LIN {X 0,Y 411.222,Z 389.379,A -85,B 0,C 180,E1 -10484.622,E2 -10484.622} C_VEL
LIN {X 0,Y 411.796,Z 392.619,A -85,B 0,C 180,E1 -10487.213,E2 -10487.213} C_VEL
LIN {X 0,Y 412.5,Z 396.68,A -85,B 0,C 180,E1 -10490.059,E2 -10490.059} C_VEL
LIN {X 0,Y 413.335,Z 401.503,A -85,B 0,C 180,E1 -10493.05,E2 -10493.05} C_VEL
LIN {X 0,Y 413.268,Z 404.546,A -85,B 0,C 180,E1 -10494.715,E2 -10494.715} C_VEL
LIN {X 0,Y 412.637,Z 410.141,A -85,B 0,C 180,E1 -10497.559,E2 -10497.559} C_VEL
LIN {X 0,Y 411.855,Z 417.317,A -85,B 0,C 180,E1 -10500.96,E2 -10500.96} C_VEL
LIN {X 0,Y 411.43,Z 424.49,A -85,B 0,C 180,E1 -10504.182,E2 -10504.182} C_VEL
LIN {X 0,Y 410.913,Z 433.22,A -85,B 0,C 180,E1 -10507.902,E2 -10507.902} C_VEL
LIN {X 0,Y 410.581,Z 440.827,A -85,B 0,C 180,E1 -10511.025,E2 -10511.025} C_VEL
LIN {X 0,Y 410.449,Z 443.604,A -85,B 0,C 180,E1 -10512.147,E2 -10512.147} C_VEL
LIN {X 0,Y 412.936,Z 457.87,A -85,B 0,C 180,E1 -10512.764,E2 -10512.764} C_VEL
LIN {X 0,Y 414.283,Z 471.211,A -85,B 0,C 180,E1 -10513.496,E2 -10513.496} C_VEL
LIN {X 0,Y 414.496,Z 479.224,A -85,B 0,C 180,E1 -10514.011,E2 -10514.011} C_VEL
LIN {X 0,Y 413.649,Z 490.528,A -85,B 0,C 180,E1 -10514.861,E2 -10514.861} C_VEL
LIN {X 0,Y 412.726,Z 502.13,A -85,B 0,C 180,E1 -10515.961,E2 -10515.961} C_VEL
LIN {X 0,Y 412.087,Z 510.937,A -85,B 0,C 180,E1 -10516.988,E2 -10516.988} C_VEL
LIN {X 0,Y 411.502,Z 519.45,A -85,B 0,C 180,E1 -10518.178,E2 -10518.178} C_VEL
LIN {X 0,Y 410.835,Z 528.113,A -85,B 0,C 180,E1 -10519.656,E2 -10519.656} C_VEL
LIN {X 0,Y 410.451,Z 535.1,A -85,B 0,C 180,E1 -10521.139,E2 -10521.139} C_VEL
LIN {X 0,Y 410.181,Z 540.719,A -85,B 0,C 180,E1 -10522.621,E2 -10522.621} C_VEL
LIN {X 0,Y 410.036,Z 545.145,A -85,B 0,C 180,E1 -10524.101,E2 -10524.101} C_VEL
LIN {X 0,Y 410.055,Z 547.506,A -85,B 0,C 180,E1 -10525.088,E2 -10525.088} C_VEL
LIN {X 0,Y 409.968,Z 549.385,A -85,B 0,C 180,E1 -10526.072,E2 -10526.072} C_VEL
LIN {X 0,Y 410.023,Z 550.818,A -85,B 0,C 180,E1 -10527.056,E2 -10527.056} C_VEL
LIN {X 0,Y 410.057,Z 551.847,A -85,B 0,C 180,E1 -10528.039,E2 -10528.039} C_VEL
LIN {X 0,Y 410.027,Z 552.471,A -85,B 0,C 180,E1 -10529.022,E2 -10529.022} C_VEL
LIN {X 0,Y 410.034,Z 552.654,A -85,B 0,C 180,E1 -10530.004,E2 -10530.004} C_VEL
LIN {X 0,Y 410.028,Z 552.419,A -85,B 0,C 180,E1 -10530.986,E2 -10530.986} C_VEL
LIN {X 0,Y 410.06,Z 551.791,A -85,B 0,C 180,E1 -10531.968,E2 -10531.968} C_VEL
LIN {X 0,Y 410.055,Z 550.757,A -85,B 0,C 180,E1 -10532.951,E2 -10532.951} C_VEL
LIN {X 0,Y 409.972,Z 549.254,A -85,B 0,C 180,E1 -10533.935,E2 -10533.935} C_VEL
LIN {X 0,Y 410.073,Z 546.197,A -85,B 0,C 180,E1 -10535.412,E2 -10535.412} C_VEL
LIN {X 0,Y 410.168,Z 542.052,A -85,B 0,C 180,E1 -10536.892,E2 -10536.892} C_VEL
LIN {X 0,Y 410.399,Z 535.69,A -85,B 0,C 180,E1 -10538.621,E2 -10538.621} C_VEL
LIN {X 0,Y 410.756,Z 528.758,A -85,B 0,C 180,E1 -10540.104,E2 -10540.104} C_VEL
LIN {X 0,Y 411.348,Z 520.088,A -85,B 0,C 180,E1 -10541.584,E2 -10541.584} C_VEL
LIN {X 0,Y 411.937,Z 511.205,A -85,B 0,C 180,E1 -10542.817,E2 -10542.817} C_VEL
LIN {X 0,Y 412.67,Z 500.31,A -85,B 0,C 180,E1 -10544.048,E2 -10544.048} C_VEL
LIN {X 0,Y 413.369,Z 489.363,A -85,B 0,C 180,E1 -10545.03,E2 -10545.03} C_VEL
LIN {X 0,Y 414.185,Z 477.508,A -85,B 0,C 180,E1 -10545.866,E2 -10545.866} C_VEL
LIN {X 0,Y 414.152,Z 473.913,A -85,B 0,C 180,E1 -10546.087,E2 -10546.087} C_VEL
LIN {X 0,Y 412.627,Z 460.357,A -85,B 0,C 180,E1 -10546.818,E2 -10546.818} C_VEL
LIN {X 0,Y 410.639,Z 447.133,A -85,B 0,C 180,E1 -10547.336,E2 -10547.336} C_VEL
LIN {X 0,Y 410.476,Z 445.601,A -85,B 0,C 180,E1 -10547.387,E2 -10547.387} C_VEL
LIN {X 0,Y 410.779,Z 437.879,A -85,B 0,C 180,E1 -10550.535,E2 -10550.535} C_VEL
LIN {X 0,Y 411.171,Z 430.287,A -85,B 0,C 180,E1 -10553.686,E2 -10553.686} C_VEL
LIN {X 0,Y 411.619,Z 422.72,A -85,B 0,C 180,E1 -10556.887,E2 -10556.887} C_VEL
LIN {X 0,Y 412.336,Z 413.826,A -85,B 0,C 180,E1 -10560.756,E2 -10560.756} C_VEL
LIN {X 0,Y 413.02,Z 406.24,A -85,B 0,C 180,E1 -10564.165,E2 -10564.165} C_VEL
LIN {X 0,Y 413.217,Z 401.187,A -85,B 0,C 180,E1 -10566.536,E2 -10566.536} C_VEL
LIN {X 0,Y 412.171,Z 394.541,A -85,B 0,C 180,E1 -10569.887,E2 -10569.887} C_VEL
LIN {X 0,Y 411.214,Z 389.263,A -85,B 0,C 180,E1 -10572.748,E2 -10572.748} C_VEL
LIN {X 0,Y 411.178,Z 389.268,A -85,B 0,C 180,E1 -10575.883,E2 -10575.883} C_VEL
LIN {X 0,Y 411.163,Z 389.271,A -85,B 0,C 180,E1 -10578.775,E2 -10578.775} C_VEL
LIN {X 0,Y 411.199,Z 389.263,A -85,B 0,C 180,E1 -10582.026,E2 -10582.026} C_VEL
LIN {X 0,Y 411.216,Z 389.265,A -85,B 0,C 180,E1 -10585.124,E2 -10585.124} C_VEL
LIN {X 0,Y 411.178,Z 389.266,A -85,B 0,C 180,E1 -10588.003,E2 -10588.003} C_VEL
LIN {X 0,Y 411.207,Z 389.265,A -85,B 0,C 180,E1 -10591.408,E2 -10591.408} C_VEL
LIN {X 0,Y 411.231,Z 389.263,A -85,B 0,C 180,E1 -10594.933,E2 -10594.933} C_VEL
LIN {X 0,Y 411.218,Z 389.26,A -85,B 0,C 180,E1 -10597.913,E2 -10597.913} C_VEL
LIN {X 0,Y 411.233,Z 389.262,A -85,B 0,C 180,E1 -10601.051,E2 -10601.051} C_VEL
LIN {X 0,Y 411.266,Z 389.255,A -85,B 0,C 180,E1 -10604.131,E2 -10604.131} C_VEL
LIN {X 0,Y 411.316,Z 389.251,A -85,B 0,C 180,E1 -10607.165,E2 -10607.165} C_VEL
LIN {X 0,Y 411.301,Z 389.25,A -85,B 0,C 180,E1 -10610.161,E2 -10610.161} C_VEL
LIN {X 0,Y 411.446,Z 389.236,A -85,B 0,C 180,E1 -10613.132,E2 -10613.132} C_VEL
LIN {X 0,Y 411.314,Z 389.252,A -85,B 0,C 180,E1 -10615.098,E2 -10615.098} C_VEL
LIN {X 0,Y 411.521,Z 389.223,A -85,B 0,C 180,E1 -10618.042,E2 -10618.042} C_VEL
LIN {X 0,Y 411.647,Z 389.208,A -85,B 0,C 180,E1 -10619.999,E2 -10619.999} C_VEL
LIN {X 0,Y 411.457,Z 389.235,A -85,B 0,C 180,E1 -10622.936,E2 -10622.936} C_VEL
LIN {X 0,Y 411.402,Z 389.239,A -85,B 0,C 180,E1 -10626.56,E2 -10626.56} C_VEL
LIN {X 0,Y 411.328,Z 389.25,A -85,B 0,C 180,E1 -10628.845,E2 -10628.845} C_VEL
LIN {X 0,Y 411.291,Z 389.251,A -85,B 0,C 180,E1 -10631.832,E2 -10631.832} C_VEL
LIN {X 0,Y 411.268,Z 389.259,A -85,B 0,C 180,E1 -10634.851,E2 -10634.851} C_VEL
LIN {X 0,Y 411.255,Z 389.257,A -85,B 0,C 180,E1 -10637.914,E2 -10637.914} C_VEL
LIN {X 0,Y 411.205,Z 389.265,A -85,B 0,C 180,E1 -10641.033,E2 -10641.033} C_VEL
LIN {X 0,Y 411.221,Z 389.262,A -85,B 0,C 180,E1 -10644.215,E2 -10644.215} C_VEL
LIN {X 0,Y 411.266,Z 389.254,A -85,B 0,C 180,E1 -10647.476,E2 -10647.476} C_VEL
LIN {X 0,Y 411.197,Z 389.267,A -85,B 0,C 180,E1 -10650.846,E2 -10650.846} C_VEL
LIN {X 0,Y 411.213,Z 389.264,A -85,B 0,C 180,E1 -10654.332,E2 -10654.332} C_VEL
LIN {X 0,Y 411.195,Z 389.265,A -85,B 0,C 180,E1 -10657.972,E2 -10657.972} C_VEL
LIN {X 0,Y 411.164,Z 389.269,A -85,B 0,C 180,E1 -10661.225,E2 -10661.225} C_VEL
LIN {X 0,Y 411.181,Z 389.27,A -85,B 0,C 180,E1 -10664.488,E2 -10664.488} C_VEL
LIN {X 0,Y 411.177,Z 389.268,A -85,B 0,C 180,E1 -10668.191,E2 -10668.191} C_VEL
LIN {X 0,Y 411.212,Z 389.265,A -85,B 0,C 180,E1 -10670.772,E2 -10670.772} C_VEL
LIN {X 0,Y 411.202,Z 389.266,A -85,B 0,C 180,E1 -10674.469,E2 -10674.469} C_VEL
LIN {X 0,Y 411.211,Z 389.263,A -85,B 0,C 180,E1 -10676.871,E2 -10676.871} C_VEL
LIN {X 0,Y 411.235,Z 389.261,A -85,B 0,C 180,E1 -10680.641,E2 -10680.641} C_VEL
LIN {X 0,Y 411.24,Z 389.259,A -85,B 0,C 180,E1 -10683.616,E2 -10683.616} C_VEL
LIN {X 0,Y 411.204,Z 389.265,A -85,B 0,C 180,E1 -10686.849,E2 -10686.849} C_VEL
LIN {X 0,Y 411.215,Z 389.264,A -85,B 0,C 180,E1 -10690.047,E2 -10690.047} C_VEL
LIN {X 0,Y 411.262,Z 389.255,A -85,B 0,C 180,E1 -10693.128,E2 -10693.128} C_VEL
LIN {X 0,Y 411.303,Z 389.25,A -85,B 0,C 180,E1 -10696.893,E2 -10696.893} C_VEL
LIN {X 0,Y 411.29,Z 389.255,A -85,B 0,C 180,E1 -10700.158,E2 -10700.158} C_VEL
LIN {X 0,Y 411.447,Z 389.233,A -85,B 0,C 180,E1 -10703.129,E2 -10703.129} C_VEL
LIN {X 0,Y 411.303,Z 389.25,A -85,B 0,C 180,E1 -10705.095,E2 -10705.095} C_VEL
LIN {X 0,Y 411.506,Z 389.228,A -85,B 0,C 180,E1 -10708.039,E2 -10708.039} C_VEL
LIN {X 0,Y 411.633,Z 389.213,A -85,B 0,C 180,E1 -10709.996,E2 -10709.996} C_VEL
LIN {X 0,Y 411.456,Z 389.231,A -85,B 0,C 180,E1 -10712.934,E2 -10712.934} C_VEL
LIN {X 0,Y 411.45,Z 389.232,A -85,B 0,C 180,E1 -10716.863,E2 -10716.863} C_VEL
LIN {X 0,Y 411.297,Z 389.254,A -85,B 0,C 180,E1 -10719.835,E2 -10719.835} C_VEL
LIN {X 0,Y 411.281,Z 389.253,A -85,B 0,C 180,E1 -10723.301,E2 -10723.301} C_VEL
LIN {X 0,Y 411.247,Z 389.257,A -85,B 0,C 180,E1 -10726.885,E2 -10726.885} C_VEL
LIN {X 0,Y 411.226,Z 389.26,A -85,B 0,C 180,E1 -10727.567,E2 -10727.567} C_VEL
LIN {X 0,Y 410.561,Z 389.346,A -85,B 0,C 180,E1 -10728.385,E2 -10728.385} C_VEL
LIN {X 0,Y 407.673,Z 389.706,A -85,B 0,C 180,E1 -10729.713,E2 -10729.713} C_VEL
LIN {X 0,Y 405.23,Z 390.007,A -85,B 0,C 180,E1 -10730.786,E2 -10730.786} C_VEL
LIN {X 0,Y 404.194,Z 390.138,A -85,B 0,C 180,E1 -10731.616,E2 -10731.616} C_VEL
LIN {X 0,Y 404.118,Z 390.144,A -85,B 0,C 180,E1 -10731.897,E2 -10731.897} C_VEL
LIN {X 0,Y 404.129,Z 390.144,A -85,B 0,C 180,E1 -10735.273,E2 -10735.273} C_VEL
LIN {X 0,Y 403.933,Z 390.172,A -85,B 0,C 180,E1 -10738.014,E2 -10738.014} C_VEL
LIN {X 0,Y 403.533,Z 390.225,A -85,B 0,C 180,E1 -10741.42,E2 -10741.42} C_VEL
LIN {X 0,Y 403.366,Z 390.535,A -85,B 0,C 180,E1 -10742.687,E2 -10742.687} C_VEL
LIN {X 0,Y 403.282,Z 394.125,A -85,B 0,C 180,E1 -10746.33,E2 -10746.33} C_VEL
LIN {X 0,Y 403.206,Z 397.745,A -85,B 0,C 180,E1 -10749.923,E2 -10749.923} C_VEL
LIN {X 0,Y 403.134,Z 400.84,A -85,B 0,C 180,E1 -10752.93,E2 -10752.93} C_VEL
LIN {X 0,Y 403.139,Z 402.439,A -85,B 0,C 180,E1 -10754.466,E2 -10754.466} C_VEL
LIN {X 0,Y 406.744,Z 417.81,A -85,B 0,C 180,E1 -10755.208,E2 -10755.208} C_VEL
LIN {X 0,Y 408.175,Z 425.22,A -85,B 0,C 180,E1 -10755.651,E2 -10755.651} C_VEL
LIN {X 0,Y 407.539,Z 438.082,A -85,B 0,C 180,E1 -10756.481,E2 -10756.481} C_VEL
LIN {X 0,Y 406.786,Z 449.886,A -85,B 0,C 180,E1 -10757.473,E2 -10757.473} C_VEL
LIN {X 0,Y 406.045,Z 460.272,A -85,B 0,C 180,E1 -10758.569,E2 -10758.569} C_VEL
LIN {X 0,Y 405.362,Z 470.406,A -85,B 0,C 180,E1 -10759.891,E2 -10759.891} C_VEL
LIN {X 0,Y 404.616,Z 479.646,A -85,B 0,C 180,E1 -10761.402,E2 -10761.402} C_VEL
LIN {X 0,Y 404.11,Z 486.882,A -85,B 0,C 180,E1 -10762.87,E2 -10762.87} C_VEL
LIN {X 0,Y 403.667,Z 492.658,A -85,B 0,C 180,E1 -10764.322,E2 -10764.322} C_VEL
LIN {X 0,Y 403.332,Z 498.17,A -85,B 0,C 180,E1 -10766.112,E2 -10766.112} C_VEL
LIN {X 0,Y 403.144,Z 502.087,A -85,B 0,C 180,E1 -10767.881,E2 -10767.881} C_VEL
LIN {X 0,Y 402.882,Z 504.621,A -85,B 0,C 180,E1 -10769.611,E2 -10769.611} C_VEL
LIN {X 0,Y 402.866,Z 505.611,A -85,B 0,C 180,E1 -10770.762,E2 -10770.762} C_VEL
LIN {X 0,Y 402.836,Z 506.055,A -85,B 0,C 180,E1 -10771.899,E2 -10771.899} C_VEL
LIN {X 0,Y 402.844,Z 506.017,A -85,B 0,C 180,E1 -10773.027,E2 -10773.027} C_VEL
LIN {X 0,Y 402.925,Z 505.42,A -85,B 0,C 180,E1 -10774.148,E2 -10774.148} C_VEL
LIN {X 0,Y 403.022,Z 504.37,A -85,B 0,C 180,E1 -10775.26,E2 -10775.26} C_VEL
LIN {X 0,Y 403.182,Z 502.794,A -85,B 0,C 180,E1 -10776.365,E2 -10776.365} C_VEL
LIN {X 0,Y 403.485,Z 499.482,A -85,B 0,C 180,E1 -10778.008,E2 -10778.008} C_VEL
LIN {X 0,Y 403.817,Z 494.983,A -85,B 0,C 180,E1 -10779.631,E2 -10779.631} C_VEL
LIN {X 0,Y 404.284,Z 489.17,A -85,B 0,C 180,E1 -10781.241,E2 -10781.241} C_VEL
LIN {X 0,Y 404.982,Z 481.767,A -85,B 0,C 180,E1 -10782.843,E2 -10782.843} C_VEL
LIN {X 0,Y 405.771,Z 472.531,A -85,B 0,C 180,E1 -10784.428,E2 -10784.428} C_VEL
LIN {X 0,Y 406.59,Z 463.669,A -85,B 0,C 180,E1 -10785.655,E2 -10785.655} C_VEL
LIN {X 0,Y 407.379,Z 453.617,A -85,B 0,C 180,E1 -10786.787,E2 -10786.787} C_VEL
LIN {X 0,Y 408.236,Z 442.106,A -85,B 0,C 180,E1 -10787.826,E2 -10787.826} C_VEL
LIN {X 0,Y 409.002,Z 430.403,A -85,B 0,C 180,E1 -10788.654,E2 -10788.654} C_VEL
LIN {X 0,Y 408.992,Z 425.264,A -85,B 0,C 180,E1 -10788.967,E2 -10788.967} C_VEL
LIN {X 0,Y 406.264,Z 413.927,A -85,B 0,C 180,E1 -10789.676,E2 -10789.676} C_VEL
LIN {X 0,Y 403.487,Z 404.713,A -85,B 0,C 180,E1 -10790.192,E2 -10790.192} C_VEL
LIN {X 0,Y 403.71,Z 401.288,A -85,B 0,C 180,E1 -10794.005,E2 -10794.005} C_VEL
LIN {X 0,Y 403.728,Z 399.563,A -85,B 0,C 180,E1 -10796.008,E2 -10796.008} C_VEL
LIN {X 0,Y 404.089,Z 396.193,A -85,B 0,C 180,E1 -10800.001,E2 -10800.001} C_VEL
LIN {X 0,Y 404.245,Z 395.339,A -85,B 0,C 180,E1 -10800.997,E2 -10800.997} C_VEL
LIN {X 0,Y 404.385,Z 391.459,A -85,B 0,C 180,E1 -10805.986,E2 -10805.986} C_VEL
LIN {X 0,Y 404.308,Z 390.129,A -85,B 0,C 180,E1 -10807.994,E2 -10807.994} C_VEL
LIN {X 0,Y 404.244,Z 390.132,A -85,B 0,C 180,E1 -10811.026,E2 -10811.026} C_VEL
LIN {X 0,Y 404.185,Z 390.139,A -85,B 0,C 180,E1 -10814.09,E2 -10814.09} C_VEL
LIN {X 0,Y 404.215,Z 390.135,A -85,B 0,C 180,E1 -10817.193,E2 -10817.193} C_VEL
LIN {X 0,Y 404.175,Z 390.141,A -85,B 0,C 180,E1 -10820.352,E2 -10820.352} C_VEL
LIN {X 0,Y 404.153,Z 390.144,A -85,B 0,C 180,E1 -10823.576,E2 -10823.576} C_VEL
LIN {X 0,Y 404.166,Z 390.143,A -85,B 0,C 180,E1 -10826.88,E2 -10826.88} C_VEL
LIN {X 0,Y 404.124,Z 390.146,A -85,B 0,C 180,E1 -10830.288,E2 -10830.288} C_VEL
LIN {X 0,Y 404.118,Z 390.147,A -85,B 0,C 180,E1 -10833.816,E2 -10833.816} C_VEL
LIN {X 0,Y 404.115,Z 390.148,A -85,B 0,C 180,E1 -10836.88,E2 -10836.88} C_VEL
LIN {X 0,Y 404.145,Z 390.145,A -85,B 0,C 180,E1 -10840.087,E2 -10840.087} C_VEL
LIN {X 0,Y 404.177,Z 390.142,A -85,B 0,C 180,E1 -10843.095,E2 -10843.095} C_VEL
LIN {X 0,Y 404.196,Z 390.36,A -85,B 0,C 180,E1 -10844.068,E2 -10844.068} C_VEL
LIN {X 0,Y 404.794,Z 393.632,A -85,B 0,C 180,E1 -10846.82,E2 -10846.82} C_VEL
LIN {X 0,Y 405.583,Z 398.22,A -85,B 0,C 180,E1 -10850.129,E2 -10850.129} C_VEL
LIN {X 0,Y 406.281,Z 402.362,A -85,B 0,C 180,E1 -10852.745,E2 -10852.745} C_VEL
LIN {X 0,Y 406.355,Z 405.193,A -85,B 0,C 180,E1 -10854.379,E2 -10854.379} C_VEL
LIN {X 0,Y 405.622,Z 411.222,A -85,B 0,C 180,E1 -10857.518,E2 -10857.518} C_VEL
LIN {X 0,Y 404.824,Z 418.276,A -85,B 0,C 180,E1 -10860.921,E2 -10860.921} C_VEL
LIN {X 0,Y 404.355,Z 425.515,A -85,B 0,C 180,E1 -10864.25,E2 -10864.25} C_VEL
LIN {X 0,Y 403.836,Z 434.203,A -85,B 0,C 180,E1 -10868.032,E2 -10868.032} C_VEL
LIN {X 0,Y 403.483,Z 441.762,A -85,B 0,C 180,E1 -10871.206,E2 -10871.206} C_VEL
LIN {X 0,Y 403.41,Z 443.174,A -85,B 0,C 180,E1 -10871.785,E2 -10871.785} C_VEL
LIN {X 0,Y 405.975,Z 457.317,A -85,B 0,C 180,E1 -10872.405,E2 -10872.405} C_VEL
LIN {X 0,Y 407.331,Z 470.431,A -85,B 0,C 180,E1 -10873.142,E2 -10873.142} C_VEL
LIN {X 0,Y 407.68,Z 479.312,A -85,B 0,C 180,E1 -10873.736,E2 -10873.736} C_VEL
LIN {X 0,Y 406.677,Z 491.865,A -85,B 0,C 180,E1 -10874.724,E2 -10874.724} C_VEL
LIN {X 0,Y 405.729,Z 503.121,A -85,B 0,C 180,E1 -10875.842,E2 -10875.842} C_VEL
LIN {X 0,Y 405.047,Z 512.296,A -85,B 0,C 180,E1 -10876.968,E2 -10876.968} C_VEL
LIN {X 0,Y 404.412,Z 520.76,A -85,B 0,C 180,E1 -10878.222,E2 -10878.222} C_VEL
LIN {X 0,Y 403.739,Z 529.089,A -85,B 0,C 180,E1 -10879.726,E2 -10879.726} C_VEL
LIN {X 0,Y 403.34,Z 535.833,A -85,B 0,C 180,E1 -10881.234,E2 -10881.234} C_VEL
LIN {X 0,Y 403.074,Z 541.994,A -85,B 0,C 180,E1 -10882.993,E2 -10882.993} C_VEL
LIN {X 0,Y 402.939,Z 546.023,A -85,B 0,C 180,E1 -10884.499,E2 -10884.499} C_VEL
LIN {X 0,Y 402.887,Z 549.004,A -85,B 0,C 180,E1 -10886.003,E2 -10886.003} C_VEL
LIN {X 0,Y 402.922,Z 550.43,A -85,B 0,C 180,E1 -10887.004,E2 -10887.004} C_VEL
LIN {X 0,Y 402.984,Z 551.453,A -85,B 0,C 180,E1 -10888.005,E2 -10888.005} C_VEL
LIN {X 0,Y 402.95,Z 552.07,A -85,B 0,C 180,E1 -10889.004,E2 -10889.004} C_VEL
LIN {X 0,Y 402.953,Z 552.239,A -85,B 0,C 180,E1 -10890.004,E2 -10890.004} C_VEL
LIN {X 0,Y 402.95,Z 551.998,A -85,B 0,C 180,E1 -10891.003,E2 -10891.003} C_VEL
LIN {X 0,Y 402.988,Z 551.362,A -85,B 0,C 180,E1 -10892.002,E2 -10892.002} C_VEL
LIN {X 0,Y 402.955,Z 550.314,A -85,B 0,C 180,E1 -10893.003,E2 -10893.003} C_VEL
LIN {X 0,Y 402.892,Z 548.795,A -85,B 0,C 180,E1 -10894.005,E2 -10894.005} C_VEL
LIN {X 0,Y 402.97,Z 545.715,A -85,B 0,C 180,E1 -10895.508,E2 -10895.508} C_VEL
LIN {X 0,Y 403.08,Z 541.545,A -85,B 0,C 180,E1 -10897.014,E2 -10897.014} C_VEL
LIN {X 0,Y 403.35,Z 535.158,A -85,B 0,C 180,E1 -10898.773,E2 -10898.773} C_VEL
LIN {X 0,Y 403.708,Z 528.192,A -85,B 0,C 180,E1 -10900.282,E2 -10900.282} C_VEL
LIN {X 0,Y 404.361,Z 519.472,A -85,B 0,C 180,E1 -10901.787,E2 -10901.787} C_VEL
LIN {X 0,Y 405.094,Z 509.107,A -85,B 0,C 180,E1 -10903.226,E2 -10903.226} C_VEL
LIN {X 0,Y 405.807,Z 498.299,A -85,B 0,C 180,E1 -10904.419,E2 -10904.419} C_VEL
LIN {X 0,Y 406.626,Z 487.004,A -85,B 0,C 180,E1 -10905.414,E2 -10905.414} C_VEL
LIN {X 0,Y 407.316,Z 476.778,A -85,B 0,C 180,E1 -10906.13,E2 -10906.13} C_VEL
LIN {X 0,Y 406.271,Z 465.644,A -85,B 0,C 180,E1 -10906.798,E2 -10906.798} C_VEL
LIN {X 0,Y 404.578,Z 452.694,A -85,B 0,C 180,E1 -10907.394,E2 -10907.394} C_VEL
LIN {X 0,Y 403.411,Z 445.239,A -85,B 0,C 180,E1 -10907.672,E2 -10907.672} C_VEL
LIN {X 0,Y 403.747,Z 437.475,A -85,B 0,C 180,E1 -10910.91,E2 -10910.91} C_VEL
LIN {X 0,Y 404.157,Z 429.886,A -85,B 0,C 180,E1 -10914.123,E2 -10914.123} C_VEL
LIN {X 0,Y 404.686,Z 421.74,A -85,B 0,C 180,E1 -10917.662,E2 -10917.662} C_VEL
LIN {X 0,Y 405.388,Z 413.487,A -85,B 0,C 180,E1 -10921.342,E2 -10921.342} C_VEL
LIN {X 0,Y 406.149,Z 405.933,A -85,B 0,C 180,E1 -10924.825,E2 -10924.825} C_VEL
LIN {X 0,Y 406.202,Z 402.199,A -85,B 0,C 180,E1 -10926.622,E2 -10926.622} C_VEL
LIN {X 0,Y 405.181,Z 395.773,A -85,B 0,C 180,E1 -10929.928,E2 -10929.928} C_VEL
LIN {X 0,Y 404.181,Z 390.139,A -85,B 0,C 180,E1 -10933.087,E2 -10933.087} C_VEL
LIN {X 0,Y 404.159,Z 390.143,A -85,B 0,C 180,E1 -10935.927,E2 -10935.927} C_VEL
LIN {X 0,Y 404.118,Z 390.148,A -85,B 0,C 180,E1 -10938.634,E2 -10938.634} C_VEL
LIN {X 0,Y 404.154,Z 390.143,A -85,B 0,C 180,E1 -10941.496,E2 -10941.496} C_VEL
LIN {X 0,Y 404.188,Z 390.139,A -85,B 0,C 180,E1 -10944.983,E2 -10944.983} C_VEL
LIN {X 0,Y 404.152,Z 390.142,A -85,B 0,C 180,E1 -10948.443,E2 -10948.443} C_VEL
LIN {X 0,Y 404.17,Z 390.142,A -85,B 0,C 180,E1 -10950.863,E2 -10950.863} C_VEL
LIN {X 0,Y 404.158,Z 390.139,A -85,B 0,C 180,E1 -10954.231,E2 -10954.231} C_VEL
LIN {X 0,Y 404.182,Z 390.138,A -85,B 0,C 180,E1 -10957.508,E2 -10957.508} C_VEL
LIN {X 0,Y 404.176,Z 390.141,A -85,B 0,C 180,E1 -10960.707,E2 -10960.707} C_VEL
LIN {X 0,Y 404.234,Z 390.131,A -85,B 0,C 180,E1 -10963.848,E2 -10963.848} C_VEL
LIN {X 0,Y 404.297,Z 390.127,A -85,B 0,C 180,E1 -10966.939,E2 -10966.939} C_VEL
LIN {X 0,Y 404.267,Z 390.126,A -85,B 0,C 180,E1 -10969.988,E2 -10969.988} C_VEL
LIN {X 0,Y 404.396,Z 390.114,A -85,B 0,C 180,E1 -10973.012,E2 -10973.012} C_VEL
LIN {X 0,Y 404.285,Z 390.128,A -85,B 0,C 180,E1 -10975.013,E2 -10975.013} C_VEL
LIN {X 0,Y 404.49,Z 390.098,A -85,B 0,C 180,E1 -10978.008,E2 -10978.008} C_VEL
LIN {X 0,Y 404.616,Z 390.083,A -85,B 0,C 180,E1 -10979.999,E2 -10979.999} C_VEL
LIN {X 0,Y 404.416,Z 390.111,A -85,B 0,C 180,E1 -10982.988,E2 -10982.988} C_VEL
LIN {X 0,Y 404.354,Z 390.116,A -85,B 0,C 180,E1 -10986.556,E2 -10986.556} C_VEL
LIN {X 0,Y 404.275,Z 390.129,A -85,B 0,C 180,E1 -10989,E2 -10989} C_VEL
LIN {X 0,Y 404.265,Z 390.127,A -85,B 0,C 180,E1 -10992.04,E2 -10992.04} C_VEL
LIN {X 0,Y 404.214,Z 390.135,A -85,B 0,C 180,E1 -10995.117,E2 -10995.117} C_VEL
LIN {X 0,Y 404.214,Z 390.135,A -85,B 0,C 180,E1 -10998.237,E2 -10998.237} C_VEL
LIN {X 0,Y 404.147,Z 390.142,A -85,B 0,C 180,E1 -11001.418,E2 -11001.418} C_VEL
LIN {X 0,Y 404.179,Z 390.141,A -85,B 0,C 180,E1 -11004.664,E2 -11004.664} C_VEL
LIN {X 0,Y 404.202,Z 390.134,A -85,B 0,C 180,E1 -11007.998,E2 -11007.998} C_VEL
LIN {X 0,Y 404.147,Z 390.141,A -85,B 0,C 180,E1 -11011.556,E2 -11011.556} C_VEL
LIN {X 0,Y 404.191,Z 390.138,A -85,B 0,C 180,E1 -11015.014,E2 -11015.014} C_VEL
LIN {X 0,Y 404.153,Z 390.145,A -85,B 0,C 180,E1 -11018.756,E2 -11018.756} C_VEL
LIN {X 0,Y 404.123,Z 390.145,A -85,B 0,C 180,E1 -11021.596,E2 -11021.596} C_VEL
LIN {X 0,Y 404.15,Z 390.145,A -85,B 0,C 180,E1 -11024.519,E2 -11024.519} C_VEL
LIN {X 0,Y 404.137,Z 390.143,A -85,B 0,C 180,E1 -11027.292,E2 -11027.292} C_VEL
LIN {X 0,Y 404.159,Z 390.142,A -85,B 0,C 180,E1 -11029.951,E2 -11029.951} C_VEL
LIN {X 0,Y 404.14,Z 390.143,A -85,B 0,C 180,E1 -11033.123,E2 -11033.123} C_VEL
LIN {X 0,Y 404.149,Z 390.144,A -85,B 0,C 180,E1 -11036.185,E2 -11036.185} C_VEL
LIN {X 0,Y 404.148,Z 390.142,A -85,B 0,C 180,E1 -11039.712,E2 -11039.712} C_VEL
LIN {X 0,Y 404.197,Z 390.136,A -85,B 0,C 180,E1 -11043.12,E2 -11043.12} C_VEL
LIN {X 0,Y 404.178,Z 390.137,A -85,B 0,C 180,E1 -11045.331,E2 -11045.331} C_VEL
LIN {X 0,Y 404.139,Z 390.145,A -85,B 0,C 180,E1 -11048.577,E2 -11048.577} C_VEL
LIN {X 0,Y 404.209,Z 390.135,A -85,B 0,C 180,E1 -11051.759,E2 -11051.759} C_VEL
LIN {X 0,Y 404.204,Z 390.136,A -85,B 0,C 180,E1 -11054.879,E2 -11054.879} C_VEL
LIN {X 0,Y 404.254,Z 390.131,A -85,B 0,C 180,E1 -11057.955,E2 -11057.955} C_VEL
LIN {X 0,Y 404.4,Z 390.114,A -85,B 0,C 180,E1 -11062.126,E2 -11062.126} C_VEL
LIN {X 0,Y 404.414,Z 390.111,A -85,B 0,C 180,E1 -11064.011,E2 -11064.011} C_VEL
LIN {X 0,Y 404.474,Z 390.104,A -85,B 0,C 180,E1 -11068.005,E2 -11068.005} C_VEL
LIN {X 0,Y 404.602,Z 390.088,A -85,B 0,C 180,E1 -11069.996,E2 -11069.996} C_VEL
LIN {X 0,Y 404.413,Z 390.108,A -85,B 0,C 180,E1 -11072.985,E2 -11072.985} C_VEL
LIN {X 0,Y 404.401,Z 390.11,A -85,B 0,C 180,E1 -11076.984,E2 -11076.984} C_VEL
LIN {X 0,Y 404.26,Z 390.131,A -85,B 0,C 180,E1 -11080.008,E2 -11080.008} C_VEL
LIN {X 0,Y 404.252,Z 390.128,A -85,B 0,C 180,E1 -11083.208,E2 -11083.208} C_VEL
LIN {X 0,Y 404.203,Z 390.134,A -85,B 0,C 180,E1 -11087.005,E2 -11087.005} C_VEL
LIN {X 0,Y 404.146,Z 390.143,A -85,B 0,C 180,E1 -11090.348,E2 -11090.348} C_VEL
LIN {X 0,Y 404.118,Z 390.144,A -85,B 0,C 180,E1 -11091.897,E2 -11091.897} C_VEL
LIN {X 0,Y 403.479,Z 390.227,A -85,B 0,C 180,E1 -11092.729,E2 -11092.729} C_VEL
LIN {X 0,Y 400.657,Z 390.584,A -85,B 0,C 180,E1 -11094.08,E2 -11094.08} C_VEL
LIN {X 0,Y 398.229,Z 390.887,A -85,B 0,C 180,E1 -11095.172,E2 -11095.172} C_VEL
LIN {X 0,Y 397.149,Z 391.018,A -85,B 0,C 180,E1 -11096.015,E2 -11096.015} C_VEL
LIN {X 0,Y 397.041,Z 391.029,A -85,B 0,C 180,E1 -11096.301,E2 -11096.301} C_VEL
LIN {X 0,Y 396.843,Z 391.053,A -85,B 0,C 180,E1 -11098.56,E2 -11098.56} C_VEL
LIN {X 0,Y 396.43,Z 391.11,A -85,B 0,C 180,E1 -11101.687,E2 -11101.687} C_VEL
LIN {X 0,Y 396.368,Z 391.116,A -85,B 0,C 180,E1 -11102.13,E2 -11102.13} C_VEL
LIN {X 0,Y 396.3,Z 392.105,A -85,B 0,C 180,E1 -11103.542,E2 -11103.542} C_VEL
LIN {X 0,Y 396.185,Z 395.575,A -85,B 0,C 180,E1 -11107.089,E2 -11107.089} C_VEL
LIN {X 0,Y 396.134,Z 398.772,A -85,B 0,C 180,E1 -11110.283,E2 -11110.283} C_VEL
LIN {X 0,Y 396.04,Z 402.377,A -85,B 0,C 180,E1 -11113.788,E2 -11113.788} C_VEL
LIN {X 0,Y 396.086,Z 402.806,A -85,B 0,C 180,E1 -11114.198,E2 -11114.198} C_VEL
LIN {X 0,Y 399.463,Z 417.152,A -85,B 0,C 180,E1 -11114.892,E2 -11114.892} C_VEL
LIN {X 0,Y 401.26,Z 425.862,A -85,B 0,C 180,E1 -11115.423,E2 -11115.423} C_VEL
LIN {X 0,Y 400.628,Z 438.667,A -85,B 0,C 180,E1 -11116.268,E2 -11116.268} C_VEL
LIN {X 0,Y 399.882,Z 450.105,A -85,B 0,C 180,E1 -11117.247,E2 -11117.247} C_VEL
LIN {X 0,Y 399.007,Z 461.638,A -85,B 0,C 180,E1 -11118.494,E2 -11118.494} C_VEL
LIN {X 0,Y 398.449,Z 469.984,A -85,B 0,C 180,E1 -11119.607,E2 -11119.607} C_VEL
LIN {X 0,Y 397.709,Z 478.791,A -85,B 0,C 180,E1 -11121.027,E2 -11121.027} C_VEL
LIN {X 0,Y 397.131,Z 486.57,A -85,B 0,C 180,E1 -11122.594,E2 -11122.594} C_VEL
LIN {X 0,Y 396.621,Z 493.007,A -85,B 0,C 180,E1 -11124.216,E2 -11124.216} C_VEL
LIN {X 0,Y 396.293,Z 498.425,A -85,B 0,C 180,E1 -11125.992,E2 -11125.992} C_VEL
LIN {X 0,Y 396.067,Z 502.472,A -85,B 0,C 180,E1 -11127.838,E2 -11127.838} C_VEL
LIN {X 0,Y 395.867,Z 504.336,A -85,B 0,C 180,E1 -11129.014,E2 -11129.014} C_VEL
LIN {X 0,Y 395.797,Z 505.804,A -85,B 0,C 180,E1 -11130.456,E2 -11130.456} C_VEL
LIN {X 0,Y 395.748,Z 506.325,A -85,B 0,C 180,E1 -11131.349,E2 -11131.349} C_VEL
LIN {X 0,Y 395.768,Z 506.495,A -85,B 0,C 180,E1 -11132.598,E2 -11132.598} C_VEL
LIN {X 0,Y 395.788,Z 506.199,A -85,B 0,C 180,E1 -11133.647,E2 -11133.647} C_VEL
LIN {X 0,Y 395.901,Z 505.316,A -85,B 0,C 180,E1 -11134.857,E2 -11134.857} C_VEL
LIN {X 0,Y 396.021,Z 504.067,A -85,B 0,C 180,E1 -11135.911,E2 -11135.911} C_VEL
LIN {X 0,Y 396.26,Z 501.855,A -85,B 0,C 180,E1 -11137.245,E2 -11137.245} C_VEL
LIN {X 0,Y 396.56,Z 498.579,A -85,B 0,C 180,E1 -11138.698,E2 -11138.698} C_VEL
LIN {X 0,Y 396.965,Z 493.646,A -85,B 0,C 180,E1 -11140.344,E2 -11140.344} C_VEL
LIN {X 0,Y 397.56,Z 487.34,A -85,B 0,C 180,E1 -11141.98,E2 -11141.98} C_VEL
LIN {X 0,Y 398.342,Z 479.427,A -85,B 0,C 180,E1 -11143.604,E2 -11143.604} C_VEL
LIN {X 0,Y 399.074,Z 471.591,A -85,B 0,C 180,E1 -11144.899,E2 -11144.899} C_VEL
LIN {X 0,Y 399.961,Z 461.333,A -85,B 0,C 180,E1 -11146.279,E2 -11146.279} C_VEL
LIN {X 0,Y 400.853,Z 451.53,A -85,B 0,C 180,E1 -11147.341,E2 -11147.341} C_VEL
LIN {X 0,Y 401.679,Z 440.505,A -85,B 0,C 180,E1 -11148.306,E2 -11148.306} C_VEL
LIN {X 0,Y 402.409,Z 427.301,A -85,B 0,C 180,E1 -11149.201,E2 -11149.201} C_VEL
LIN {X 0,Y 399.551,Z 415.281,A -85,B 0,C 180,E1 -11150.002,E2 -11150.002} C_VEL
LIN {X 0,Y 396.444,Z 405.258,A -85,B 0,C 180,E1 -11150.573,E2 -11150.573} C_VEL
LIN {X 0,Y 396.668,Z 402.293,A -85,B 0,C 180,E1 -11153.899,E2 -11153.899} C_VEL
LIN {X 0,Y 396.694,Z 400.547,A -85,B 0,C 180,E1 -11155.937,E2 -11155.937} C_VEL
LIN {X 0,Y 397.068,Z 397.162,A -85,B 0,C 180,E1 -11160.001,E2 -11160.001} C_VEL
LIN {X 0,Y 397.1,Z 395.586,A -85,B 0,C 180,E1 -11162.029,E2 -11162.029} C_VEL
LIN {X 0,Y 397.373,Z 392.479,A -85,B 0,C 180,E1 -11166.092,E2 -11166.092} C_VEL
LIN {X 0,Y 397.278,Z 391.055,A -85,B 0,C 180,E1 -11168.137,E2 -11168.137} C_VEL
LIN {X 0,Y 397.189,Z 391.011,A -85,B 0,C 180,E1 -11171.224,E2 -11171.224} C_VEL
LIN {X 0,Y 397.15,Z 391.015,A -85,B 0,C 180,E1 -11174.345,E2 -11174.345} C_VEL
LIN {X 0,Y 397.165,Z 391.015,A -85,B 0,C 180,E1 -11177.508,E2 -11177.508} C_VEL
LIN {X 0,Y 397.125,Z 391.019,A -85,B 0,C 180,E1 -11180.73,E2 -11180.73} C_VEL
LIN {X 0,Y 397.11,Z 391.019,A -85,B 0,C 180,E1 -11184.021,E2 -11184.021} C_VEL
LIN {X 0,Y 397.165,Z 391.013,A -85,B 0,C 180,E1 -11187.393,E2 -11187.393} C_VEL
LIN {X 0,Y 397.055,Z 391.026,A -85,B 0,C 180,E1 -11190.885,E2 -11190.885} C_VEL
LIN {X 0,Y 397.099,Z 391.022,A -85,B 0,C 180,E1 -11194.497,E2 -11194.497} C_VEL
LIN {X 0,Y 397.086,Z 391.024,A -85,B 0,C 180,E1 -11198.278,E2 -11198.278} C_VEL
LIN {X 0,Y 397.133,Z 391.02,A -85,B 0,C 180,E1 -11201.997,E2 -11201.997} C_VEL
LIN {X 0,Y 397.145,Z 391.026,A -85,B 0,C 180,E1 -11203.188,E2 -11203.188} C_VEL
LIN {X 0,Y 397.796,Z 394.714,A -85,B 0,C 180,E1 -11206.454,E2 -11206.454} C_VEL
LIN {X 0,Y 398.423,Z 398.536,A -85,B 0,C 180,E1 -11209.333,E2 -11209.333} C_VEL
LIN {X 0,Y 399.229,Z 403.135,A -85,B 0,C 180,E1 -11212.39,E2 -11212.39} C_VEL
LIN {X 0,Y 399.346,Z 406.717,A -85,B 0,C 180,E1 -11214.502,E2 -11214.502} C_VEL
LIN {X 0,Y 398.502,Z 413.465,A -85,B 0,C 180,E1 -11218.062,E2 -11218.062} C_VEL
LIN {X 0,Y 397.617,Z 421.753,A -85,B 0,C 180,E1 -11222.101,E2 -11222.101} C_VEL
LIN {X 0,Y 397.192,Z 427.754,A -85,B 0,C 180,E1 -11224.876,E2 -11224.876} C_VEL
LIN {X 0,Y 396.733,Z 435.168,A -85,B 0,C 180,E1 -11228.165,E2 -11228.165} C_VEL
LIN {X 0,Y 396.393,Z 442.641,A -85,B 0,C 180,E1 -11231.36,E2 -11231.36} C_VEL
LIN {X 0,Y 399.253,Z 458.495,A -85,B 0,C 180,E1 -11232.124,E2 -11232.124} C_VEL
LIN {X 0,Y 400.579,Z 471.833,A -85,B 0,C 180,E1 -11232.915,E2 -11232.915} C_VEL
LIN {X 0,Y 400.859,Z 479.474,A -85,B 0,C 180,E1 -11233.452,E2 -11233.452} C_VEL
LIN {X 0,Y 399.831,Z 491.906,A -85,B 0,C 180,E1 -11234.456,E2 -11234.456} C_VEL
LIN {X 0,Y 398.825,Z 503.032,A -85,B 0,C 180,E1 -11235.591,E2 -11235.591} C_VEL
LIN {X 0,Y 398.067,Z 512.115,A -85,B 0,C 180,E1 -11236.735,E2 -11236.735} C_VEL
LIN {X 0,Y 397.412,Z 520.514,A -85,B 0,C 180,E1 -11238.011,E2 -11238.011} C_VEL
LIN {X 0,Y 396.699,Z 528.804,A -85,B 0,C 180,E1 -11239.542,E2 -11239.542} C_VEL
LIN {X 0,Y 396.29,Z 535.529,A -85,B 0,C 180,E1 -11241.077,E2 -11241.077} C_VEL
LIN {X 0,Y 396.001,Z 541.658,A -85,B 0,C 180,E1 -11242.868,E2 -11242.868} C_VEL
LIN {X 0,Y 395.836,Z 545.192,A -85,B 0,C 180,E1 -11244.185,E2 -11244.185} C_VEL
LIN {X 0,Y 395.808,Z 548.633,A -85,B 0,C 180,E1 -11245.931,E2 -11245.931} C_VEL
LIN {X 0,Y 395.912,Z 551.066,A -85,B 0,C 180,E1 -11247.969,E2 -11247.969} C_VEL
LIN {X 0,Y 395.875,Z 551.668,A -85,B 0,C 180,E1 -11248.987,E2 -11248.987} C_VEL
LIN {X 0,Y 395.875,Z 551.82,A -85,B 0,C 180,E1 -11250.004,E2 -11250.004} C_VEL
LIN {X 0,Y 395.875,Z 551.57,A -85,B 0,C 180,E1 -11251.021,E2 -11251.021} C_VEL
LIN {X 0,Y 395.917,Z 550.924,A -85,B 0,C 180,E1 -11252.038,E2 -11252.038} C_VEL
LIN {X 0,Y 395.856,Z 549.858,A -85,B 0,C 180,E1 -11253.057,E2 -11253.057} C_VEL
LIN {X 0,Y 395.815,Z 548.324,A -85,B 0,C 180,E1 -11254.076,E2 -11254.076} C_VEL
LIN {X 0,Y 395.873,Z 544.588,A -85,B 0,C 180,E1 -11255.862,E2 -11255.862} C_VEL
LIN {X 0,Y 396.062,Z 539.38,A -85,B 0,C 180,E1 -11257.651,E2 -11257.651} C_VEL
LIN {X 0,Y 396.413,Z 532.412,A -85,B 0,C 180,E1 -11259.442,E2 -11259.442} C_VEL
LIN {X 0,Y 396.857,Z 524.857,A -85,B 0,C 180,E1 -11260.978,E2 -11260.978} C_VEL
LIN {X 0,Y 397.502,Z 517.165,A -85,B 0,C 180,E1 -11262.253,E2 -11262.253} C_VEL
LIN {X 0,Y 398.199,Z 507.304,A -85,B 0,C 180,E1 -11263.589,E2 -11263.589} C_VEL
LIN {X 0,Y 399.003,Z 496.179,A -85,B 0,C 180,E1 -11264.801,E2 -11264.801} C_VEL
LIN {X 0,Y 399.745,Z 486.071,A -85,B 0,C 180,E1 -11265.686,E2 -11265.686} C_VEL
LIN {X 0,Y 400.271,Z 475.852,A -85,B 0,C 180,E1 -11266.411,E2 -11266.411} C_VEL
LIN {X 0,Y 398.936,Z 463.029,A -85,B 0,C 180,E1 -11267.174,E2 -11267.174} C_VEL
LIN {X 0,Y 397.031,Z 449.609,A -85,B 0,C 180,E1 -11267.77,E2 -11267.77} C_VEL
LIN {X 0,Y 396.328,Z 444.93,A -85,B 0,C 180,E1 -11267.935,E2 -11267.935} C_VEL
LIN {X 0,Y 396.711,Z 437.046,A -85,B 0,C 180,E1 -11271.298,E2 -11271.298} C_VEL
LIN {X 0,Y 397.14,Z 429.503,A -85,B 0,C 180,E1 -11274.577,E2 -11274.577} C_VEL
LIN {X 0,Y 397.679,Z 421.974,A -85,B 0,C 180,E1 -11277.916,E2 -11277.916} C_VEL
LIN {X 0,Y 398.368,Z 414.4,A -85,B 0,C 180,E1 -11281.365,E2 -11281.365} C_VEL
LIN {X 0,Y 399.138,Z 406.851,A -85,B 0,C 180,E1 -11284.911,E2 -11284.911} C_VEL
LIN {X 0,Y 399.164,Z 403.061,A -85,B 0,C 180,E1 -11286.775,E2 -11286.775} C_VEL
LIN {X 0,Y 398.18,Z 396.875,A -85,B 0,C 180,E1 -11290.009,E2 -11290.009} C_VEL
LIN {X 0,Y 397.135,Z 391.016,A -85,B 0,C 180,E1 -11293.338,E2 -11293.338} C_VEL
LIN {X 0,Y 397.112,Z 391.019,A -85,B 0,C 180,E1 -11296.523,E2 -11296.523} C_VEL
LIN {X 0,Y 397.101,Z 391.019,A -85,B 0,C 180,E1 -11300.42,E2 -11300.42} C_VEL
LIN {X 0,Y 397.11,Z 391.022,A -85,B 0,C 180,E1 -11303.005,E2 -11303.005} C_VEL
LIN {X 0,Y 397.126,Z 391.018,A -85,B 0,C 180,E1 -11306.727,E2 -11306.727} C_VEL
LIN {X 0,Y 397.132,Z 391.015,A -85,B 0,C 180,E1 -11310.296,E2 -11310.296} C_VEL
LIN {X 0,Y 397.104,Z 391.019,A -85,B 0,C 180,E1 -11313.739,E2 -11313.739} C_VEL
LIN {X 0,Y 397.117,Z 391.021,A -85,B 0,C 180,E1 -11317.085,E2 -11317.085} C_VEL
LIN {X 0,Y 397.161,Z 391.012,A -85,B 0,C 180,E1 -11320.353,E2 -11320.353} C_VEL
LIN {X 0,Y 397.18,Z 391.011,A -85,B 0,C 180,E1 -11323.553,E2 -11323.553} C_VEL
LIN {X 0,Y 397.244,Z 391.004,A -85,B 0,C 180,E1 -11326.702,E2 -11326.702} C_VEL
LIN {X 0,Y 397.228,Z 391.003,A -85,B 0,C 180,E1 -11329.808,E2 -11329.808} C_VEL
LIN {X 0,Y 397.344,Z 390.992,A -85,B 0,C 180,E1 -11332.887,E2 -11332.887} C_VEL
LIN {X 0,Y 397.256,Z 391.004,A -85,B 0,C 180,E1 -11334.924,E2 -11334.924} C_VEL
LIN {X 0,Y 397.459,Z 390.974,A -85,B 0,C 180,E1 -11337.972,E2 -11337.972} C_VEL
LIN {X 0,Y 397.586,Z 390.959,A -85,B 0,C 180,E1 -11339.999,E2 -11339.999} C_VEL
LIN {X 0,Y 397.35,Z 390.991,A -85,B 0,C 180,E1 -11343.041,E2 -11343.041} C_VEL
LIN {X 0,Y 397.31,Z 390.992,A -85,B 0,C 180,E1 -11346.55,E2 -11346.55} C_VEL
LIN {X 0,Y 397.246,Z 391.004,A -85,B 0,C 180,E1 -11349.161,E2 -11349.161} C_VEL
LIN {X 0,Y 397.229,Z 391.004,A -85,B 0,C 180,E1 -11352.257,E2 -11352.257} C_VEL
LIN {X 0,Y 397.188,Z 391.009,A -85,B 0,C 180,E1 -11355.391,E2 -11355.391} C_VEL
LIN {X 0,Y 397.167,Z 391.014,A -85,B 0,C 180,E1 -11358.572,E2 -11358.572} C_VEL
LIN {X 0,Y 397.105,Z 391.019,A -85,B 0,C 180,E1 -11361.817,E2 -11361.817} C_VEL
LIN {X 0,Y 397.16,Z 391.012,A -85,B 0,C 180,E1 -11365.51,E2 -11365.51} C_VEL
LIN {X 0,Y 397.124,Z 391.021,A -85,B 0,C 180,E1 -11368.542,E2 -11368.542} C_VEL
LIN {X 0,Y 397.086,Z 391.021,A -85,B 0,C 180,E1 -11372.07,E2 -11372.07} C_VEL
LIN {X 0,Y 397.126,Z 391.015,A -85,B 0,C 180,E1 -11375.501,E2 -11375.501} C_VEL
LIN {X 0,Y 397.11,Z 391.021,A -85,B 0,C 180,E1 -11378.854,E2 -11378.854} C_VEL
LIN {X 0,Y 397.07,Z 391.026,A -85,B 0,C 180,E1 -11382.266,E2 -11382.266} C_VEL
LIN {X 0,Y 397.092,Z 391.022,A -85,B 0,C 180,E1 -11385.066,E2 -11385.066} C_VEL
LIN {X 0,Y 397.067,Z 391.025,A -85,B 0,C 180,E1 -11388.019,E2 -11388.019} C_VEL
LIN {X 0,Y 397.129,Z 391.016,A -85,B 0,C 180,E1 -11391.137,E2 -11391.137} C_VEL
LIN {X 0,Y 397.123,Z 391.02,A -85,B 0,C 180,E1 -11394.494,E2 -11394.494} C_VEL
LIN {X 0,Y 397.081,Z 391.023,A -85,B 0,C 180,E1 -11397.925,E2 -11397.925} C_VEL
LIN {X 0,Y 397.124,Z 391.016,A -85,B 0,C 180,E1 -11401.453,E2 -11401.453} C_VEL
LIN {X 0,Y 397.155,Z 391.016,A -85,B 0,C 180,E1 -11404.484,E2 -11404.484} C_VEL
LIN {X 0,Y 397.11,Z 391.019,A -85,B 0,C 180,E1 -11407.083,E2 -11407.083} C_VEL
LIN {X 0,Y 397.148,Z 391.017,A -85,B 0,C 180,E1 -11410.35,E2 -11410.35} C_VEL
LIN {X 0,Y 397.165,Z 391.011,A -85,B 0,C 180,E1 -11413.55,E2 -11413.55} C_VEL
LIN {X 0,Y 397.226,Z 391.005,A -85,B 0,C 180,E1 -11416.699,E2 -11416.699} C_VEL
LIN {X 0,Y 397.215,Z 391.007,A -85,B 0,C 180,E1 -11419.805,E2 -11419.805} C_VEL
LIN {X 0,Y 397.345,Z 390.99,A -85,B 0,C 180,E1 -11422.884,E2 -11422.884} C_VEL
LIN {X 0,Y 397.247,Z 391.001,A -85,B 0,C 180,E1 -11424.921,E2 -11424.921} C_VEL
LIN {X 0,Y 397.443,Z 390.98,A -85,B 0,C 180,E1 -11427.97,E2 -11427.97} C_VEL
LIN {X 0,Y 397.571,Z 390.964,A -85,B 0,C 180,E1 -11429.996,E2 -11429.996} C_VEL
LIN {X 0,Y 397.372,Z 390.985,A -85,B 0,C 180,E1 -11433.038,E2 -11433.038} C_VEL
LIN {X 0,Y 397.354,Z 390.987,A -85,B 0,C 180,E1 -11437.108,E2 -11437.108} C_VEL
LIN {X 0,Y 397.217,Z 391.008,A -85,B 0,C 180,E1 -11440.187,E2 -11440.187} C_VEL
LIN {X 0,Y 397.212,Z 391.005,A -85,B 0,C 180,E1 -11443.317,E2 -11443.317} C_VEL
LIN {X 0,Y 397.156,Z 391.014,A -85,B 0,C 180,E1 -11446.443,E2 -11446.443} C_VEL
LIN {X 0,Y 397.131,Z 391.017,A -85,B 0,C 180,E1 -11449.643,E2 -11449.643} C_VEL
LIN {X 0,Y 397.116,Z 391.017,A -85,B 0,C 180,E1 -11453.037,E2 -11453.037} C_VEL
LIN {X 0,Y 397.041,Z 391.029,A -85,B 0,C 180,E1 -11456.301,E2 -11456.301} C_VEL
LIN {X 0,Y 396.299,Z 391.12,A -85,B 0,C 180,E1 -11457.147,E2 -11457.147} C_VEL
LIN {X 0,Y 393.318,Z 391.492,A -85,B 0,C 180,E1 -11458.519,E2 -11458.519} C_VEL
LIN {X 0,Y 390.778,Z 391.811,A -85,B 0,C 180,E1 -11459.627,E2 -11459.627} C_VEL
LIN {X 0,Y 389.624,Z 391.956,A -85,B 0,C 180,E1 -11460.486,E2 -11460.486} C_VEL
LIN {X 0,Y 389.495,Z 391.97,A -85,B 0,C 180,E1 -11460.777,E2 -11460.777} C_VEL
LIN {X 0,Y 389.256,Z 392.121,A -85,B 0,C 180,E1 -11462.79,E2 -11462.79} C_VEL
LIN {X 0,Y 389.115,Z 395.799,A -85,B 0,C 180,E1 -11466.58,E2 -11466.58} C_VEL
LIN {X 0,Y 389.087,Z 398.387,A -85,B 0,C 180,E1 -11469.206,E2 -11469.206} C_VEL
LIN {X 0,Y 389.013,Z 401.403,A -85,B 0,C 180,E1 -11472.209,E2 -11472.209} C_VEL
LIN {X 0,Y 388.99,Z 403.15,A -85,B 0,C 180,E1 -11473.899,E2 -11473.899} C_VEL
LIN {X 0,Y 392.599,Z 418.245,A -85,B 0,C 180,E1 -11474.663,E2 -11474.663} C_VEL
LIN {X 0,Y 394.385,Z 427.641,A -85,B 0,C 180,E1 -11475.257,E2 -11475.257} C_VEL
LIN {X 0,Y 393.657,Z 440.418,A -85,B 0,C 180,E1 -11476.14,E2 -11476.14} C_VEL
LIN {X 0,Y 392.846,Z 451.916,A -85,B 0,C 180,E1 -11477.172,E2 -11477.172} C_VEL
LIN {X 0,Y 391.978,Z 463.197,A -85,B 0,C 180,E1 -11478.442,E2 -11478.442} C_VEL
LIN {X 0,Y 391.296,Z 472.263,A -85,B 0,C 180,E1 -11479.716,E2 -11479.716} C_VEL
LIN {X 0,Y 390.524,Z 481.379,A -85,B 0,C 180,E1 -11481.292,E2 -11481.292} C_VEL
LIN {X 0,Y 389.948,Z 489.049,A -85,B 0,C 180,E1 -11482.96,E2 -11482.96} C_VEL
LIN {X 0,Y 389.461,Z 495.397,A -85,B 0,C 180,E1 -11484.73,E2 -11484.73} C_VEL
LIN {X 0,Y 389.129,Z 500.626,A -85,B 0,C 180,E1 -11486.672,E2 -11486.672} C_VEL
LIN {X 0,Y 388.855,Z 503.86,A -85,B 0,C 180,E1 -11488.391,E2 -11488.391} C_VEL
LIN {X 0,Y 388.708,Z 505.994,A -85,B 0,C 180,E1 -11490.2,E2 -11490.2} C_VEL
LIN {X 0,Y 388.682,Z 506.942,A -85,B 0,C 180,E1 -11492.363,E2 -11492.363} C_VEL
LIN {X 0,Y 388.758,Z 506.274,A -85,B 0,C 180,E1 -11494.288,E2 -11494.288} C_VEL
LIN {X 0,Y 388.876,Z 505.234,A -85,B 0,C 180,E1 -11495.44,E2 -11495.44} C_VEL
LIN {X 0,Y 389.167,Z 502.881,A -85,B 0,C 180,E1 -11497.061,E2 -11497.061} C_VEL
LIN {X 0,Y 389.535,Z 499.05,A -85,B 0,C 180,E1 -11498.849,E2 -11498.849} C_VEL
LIN {X 0,Y 389.98,Z 494.135,A -85,B 0,C 180,E1 -11500.526,E2 -11500.526} C_VEL
LIN {X 0,Y 390.616,Z 487.839,A -85,B 0,C 180,E1 -11502.191,E2 -11502.191} C_VEL
LIN {X 0,Y 391.445,Z 479.941,A -85,B 0,C 180,E1 -11503.843,E2 -11503.843} C_VEL
LIN {X 0,Y 392.323,Z 471.204,A -85,B 0,C 180,E1 -11505.296,E2 -11505.296} C_VEL
LIN {X 0,Y 393.273,Z 460.776,A -85,B 0,C 180,E1 -11506.699,E2 -11506.699} C_VEL
LIN {X 0,Y 394.305,Z 449.696,A -85,B 0,C 180,E1 -11507.878,E2 -11507.878} C_VEL
LIN {X 0,Y 395.194,Z 438.109,A -85,B 0,C 180,E1 -11508.861,E2 -11508.861} C_VEL
LIN {X 0,Y 395.663,Z 428.458,A -85,B 0,C 180,E1 -11509.518,E2 -11509.518} C_VEL
LIN {X 0,Y 393.135,Z 417.651,A -85,B 0,C 180,E1 -11510.275,E2 -11510.275} C_VEL
LIN {X 0,Y 389.429,Z 405.705,A -85,B 0,C 180,E1 -11511.013,E2 -11511.013} C_VEL
LIN {X 0,Y 389.74,Z 402.404,A -85,B 0,C 180,E1 -11514.828,E2 -11514.828} C_VEL
LIN {X 0,Y 390.047,Z 398.182,A -85,B 0,C 180,E1 -11520.001,E2 -11520.001} C_VEL
LIN {X 0,Y 390.088,Z 396.579,A -85,B 0,C 180,E1 -11522.066,E2 -11522.066} C_VEL
LIN {X 0,Y 390.362,Z 393.53,A -85,B 0,C 180,E1 -11526.202,E2 -11526.202} C_VEL
LIN {X 0,Y 390.253,Z 392.123,A -85,B 0,C 180,E1 -11528.284,E2 -11528.284} C_VEL
LIN {X 0,Y 390.137,Z 391.89,A -85,B 0,C 180,E1 -11531.43,E2 -11531.43} C_VEL
LIN {X 0,Y 390.118,Z 391.892,A -85,B 0,C 180,E1 -11534.609,E2 -11534.609} C_VEL
LIN {X 0,Y 390.111,Z 391.892,A -85,B 0,C 180,E1 -11537.835,E2 -11537.835} C_VEL
LIN {X 0,Y 390.077,Z 391.895,A -85,B 0,C 180,E1 -11541.122,E2 -11541.122} C_VEL
LIN {X 0,Y 390.054,Z 391.897,A -85,B 0,C 180,E1 -11544.483,E2 -11544.483} C_VEL
LIN {X 0,Y 390.086,Z 391.894,A -85,B 0,C 180,E1 -11548.028,E2 -11548.028} C_VEL
LIN {X 0,Y 389.999,Z 391.906,A -85,B 0,C 180,E1 -11551.507,E2 -11551.507} C_VEL
LIN {X 0,Y 390.059,Z 391.899,A -85,B 0,C 180,E1 -11555.21,E2 -11555.21} C_VEL
LIN {X 0,Y 390.072,Z 391.899,A -85,B 0,C 180,E1 -11559.095,E2 -11559.095} C_VEL
LIN {X 0,Y 390.114,Z 392.045,A -85,B 0,C 180,E1 -11562.583,E2 -11562.583} C_VEL
LIN {X 0,Y 390.765,Z 395.721,A -85,B 0,C 180,E1 -11566.007,E2 -11566.007} C_VEL
LIN {X 0,Y 391.387,Z 399.474,A -85,B 0,C 180,E1 -11568.955,E2 -11568.955} C_VEL
LIN {X 0,Y 392.275,Z 404.65,A -85,B 0,C 180,E1 -11572.479,E2 -11572.479} C_VEL
LIN {X 0,Y 392.377,Z 407.855,A -85,B 0,C 180,E1 -11574.406,E2 -11574.406} C_VEL
LIN {X 0,Y 391.592,Z 413.569,A -85,B 0,C 180,E1 -11577.515,E2 -11577.515} C_VEL
LIN {X 0,Y 390.76,Z 420.376,A -85,B 0,C 180,E1 -11580.953,E2 -11580.953} C_VEL
LIN {X 0,Y 390.235,Z 427.19,A -85,B 0,C 180,E1 -11584.223,E2 -11584.223} C_VEL
LIN {X 0,Y 389.728,Z 434.919,A -85,B 0,C 180,E1 -11587.752,E2 -11587.752} C_VEL
LIN {X 0,Y 389.345,Z 442.177,A -85,B 0,C 180,E1 -11590.942,E2 -11590.942} C_VEL
LIN {X 0,Y 392.292,Z 457.749,A -85,B 0,C 180,E1 -11591.717,E2 -11591.717} C_VEL
LIN {X 0,Y 393.618,Z 470.094,A -85,B 0,C 180,E1 -11592.469,E2 -11592.469} C_VEL
LIN {X 0,Y 394.042,Z 479.634,A -85,B 0,C 180,E1 -11593.157,E2 -11593.157} C_VEL
LIN {X 0,Y 392.988,Z 491.946,A -85,B 0,C 180,E1 -11594.178,E2 -11594.178} C_VEL
LIN {X 0,Y 391.944,Z 502.952,A -85,B 0,C 180,E1 -11595.333,E2 -11595.333} C_VEL
LIN {X 0,Y 391.107,Z 511.977,A -85,B 0,C 180,E1 -11596.495,E2 -11596.495} C_VEL
LIN {X 0,Y 390.442,Z 520.331,A -85,B 0,C 180,E1 -11597.794,E2 -11597.794} C_VEL
LIN {X 0,Y 389.679,Z 528.57,A -85,B 0,C 180,E1 -11599.351,E2 -11599.351} C_VEL
LIN {X 0,Y 389.304,Z 534.204,A -85,B 0,C 180,E1 -11600.654,E2 -11600.654} C_VEL
LIN {X 0,Y 388.983,Z 539.748,A -85,B 0,C 180,E1 -11602.216,E2 -11602.216} C_VEL
LIN {X 0,Y 388.776,Z 544.307,A -85,B 0,C 180,E1 -11603.857,E2 -11603.857} C_VEL
LIN {X 0,Y 388.766,Z 546.435,A -85,B 0,C 180,E1 -11604.818,E2 -11604.818} C_VEL
LIN {X 0,Y 388.731,Z 548.262,A -85,B 0,C 180,E1 -11605.857,E2 -11605.857} C_VEL
LIN {X 0,Y 388.84,Z 550.681,A -85,B 0,C 180,E1 -11607.932,E2 -11607.932} C_VEL
LIN {X 0,Y 388.802,Z 551.263,A -85,B 0,C 180,E1 -11608.968,E2 -11608.968} C_VEL
LIN {X 0,Y 388.8,Z 551.401,A -85,B 0,C 180,E1 -11610.004,E2 -11610.004} C_VEL
LIN {X 0,Y 388.803,Z 551.14,A -85,B 0,C 180,E1 -11611.039,E2 -11611.039} C_VEL
LIN {X 0,Y 388.847,Z 550.483,A -85,B 0,C 180,E1 -11612.075,E2 -11612.075} C_VEL
LIN {X 0,Y 388.76,Z 549.39,A -85,B 0,C 180,E1 -11613.113,E2 -11613.113} C_VEL
LIN {X 0,Y 388.739,Z 547.84,A -85,B 0,C 180,E1 -11614.151,E2 -11614.151} C_VEL
LIN {X 0,Y 388.778,Z 544.438,A -85,B 0,C 180,E1 -11615.818,E2 -11615.818} C_VEL
LIN {X 0,Y 388.936,Z 540.469,A -85,B 0,C 180,E1 -11617.27,E2 -11617.27} C_VEL
LIN {X 0,Y 389.216,Z 534.008,A -85,B 0,C 180,E1 -11619.094,E2 -11619.094} C_VEL
LIN {X 0,Y 389.64,Z 526.936,A -85,B 0,C 180,E1 -11620.658,E2 -11620.658} C_VEL
LIN {X 0,Y 390.391,Z 518.1,A -85,B 0,C 180,E1 -11622.215,E2 -11622.215} C_VEL
LIN {X 0,Y 391.04,Z 509.056,A -85,B 0,C 180,E1 -11623.515,E2 -11623.515} C_VEL
LIN {X 0,Y 391.765,Z 499.139,A -85,B 0,C 180,E1 -11624.682,E2 -11624.682} C_VEL
LIN {X 0,Y 392.627,Z 488.216,A -85,B 0,C 180,E1 -11625.711,E2 -11625.711} C_VEL
LIN {X 0,Y 393.362,Z 478.073,A -85,B 0,C 180,E1 -11626.48,E2 -11626.48} C_VEL
LIN {X 0,Y 392.309,Z 466.28,A -85,B 0,C 180,E1 -11627.241,E2 -11627.241} C_VEL
LIN {X 0,Y 390.556,Z 452.907,A -85,B 0,C 180,E1 -11627.909,E2 -11627.909} C_VEL
LIN {X 0,Y 389.296,Z 444.617,A -85,B 0,C 180,E1 -11628.216,E2 -11628.216} C_VEL
LIN {X 0,Y 389.677,Z 436.624,A -85,B 0,C 180,E1 -11631.702,E2 -11631.702} C_VEL
LIN {X 0,Y 390.16,Z 429.086,A -85,B 0,C 180,E1 -11635.047,E2 -11635.047} C_VEL
LIN {X 0,Y 390.66,Z 422.212,A -85,B 0,C 180,E1 -11638.173,E2 -11638.173} C_VEL
LIN {X 0,Y 391.327,Z 415.283,A -85,B 0,C 180,E1 -11641.391,E2 -11641.391} C_VEL
LIN {X 0,Y 392.128,Z 407.761,A -85,B 0,C 180,E1 -11645,E2 -11645} C_VEL
LIN {X 0,Y 392.127,Z 403.976,A -85,B 0,C 180,E1 -11646.902,E2 -11646.902} C_VEL
LIN {X 0,Y 391.099,Z 397.594,A -85,B 0,C 180,E1 -11650.313,E2 -11650.313} C_VEL
LIN {X 0,Y 390.075,Z 391.896,A -85,B 0,C 180,E1 -11653.609,E2 -11653.609} C_VEL
LIN {X 0,Y 390.066,Z 391.897,A -85,B 0,C 180,E1 -11656.79,E2 -11656.79} C_VEL
LIN {X 0,Y 390.024,Z 391.904,A -85,B 0,C 180,E1 -11659.556,E2 -11659.556} C_VEL
LIN {X 0,Y 390.054,Z 391.897,A -85,B 0,C 180,E1 -11662.451,E2 -11662.451} C_VEL
LIN {X 0,Y 390.076,Z 391.894,A -85,B 0,C 180,E1 -11666.045,E2 -11666.045} C_VEL
LIN {X 0,Y 390.059,Z 391.896,A -85,B 0,C 180,E1 -11669.87,E2 -11669.87} C_VEL
LIN {X 0,Y 390.066,Z 391.899,A -85,B 0,C 180,E1 -11673.227,E2 -11673.227} C_VEL
LIN {X 0,Y 390.081,Z 391.896,A -85,B 0,C 180,E1 -11676.764,E2 -11676.764} C_VEL
LIN {X 0,Y 390.118,Z 391.889,A -85,B 0,C 180,E1 -11679.983,E2 -11679.983} C_VEL
LIN {X 0,Y 390.152,Z 391.888,A -85,B 0,C 180,E1 -11683.248,E2 -11683.248} C_VEL
LIN {X 0,Y 390.21,Z 391.879,A -85,B 0,C 180,E1 -11686.561,E2 -11686.561} C_VEL
LIN {X 0,Y 390.179,Z 391.881,A -85,B 0,C 180,E1 -11689.622,E2 -11689.622} C_VEL
LIN {X 0,Y 390.293,Z 391.87,A -85,B 0,C 180,E1 -11692.758,E2 -11692.758} C_VEL
LIN {X 0,Y 390.228,Z 391.879,A -85,B 0,C 180,E1 -11694.833,E2 -11694.833} C_VEL
LIN {X 0,Y 390.428,Z 391.85,A -85,B 0,C 180,E1 -11697.936,E2 -11697.936} C_VEL
LIN {X 0,Y 390.555,Z 391.834,A -85,B 0,C 180,E1 -11699.999,E2 -11699.999} C_VEL
LIN {X 0,Y 390.286,Z 391.871,A -85,B 0,C 180,E1 -11703.096,E2 -11703.096} C_VEL
LIN {X 0,Y 390.269,Z 391.869,A -85,B 0,C 180,E1 -11706.542,E2 -11706.542} C_VEL
LIN {X 0,Y 390.203,Z 391.88,A -85,B 0,C 180,E1 -11709.328,E2 -11709.328} C_VEL
LIN {X 0,Y 390.181,Z 391.884,A -85,B 0,C 180,E1 -11712.482,E2 -11712.482} C_VEL
LIN {X 0,Y 390.149,Z 391.884,A -85,B 0,C 180,E1 -11715.675,E2 -11715.675} C_VEL
LIN {X 0,Y 390.112,Z 391.893,A -85,B 0,C 180,E1 -11718.921,E2 -11718.921} C_VEL
LIN {X 0,Y 390.047,Z 391.9,A -85,B 0,C 180,E1 -11722.233,E2 -11722.233} C_VEL
LIN {X 0,Y 390.127,Z 391.888,A -85,B 0,C 180,E1 -11725.741,E2 -11725.741} C_VEL
LIN {X 0,Y 390.061,Z 391.898,A -85,B 0,C 180,E1 -11729.108,E2 -11729.108} C_VEL
LIN {X 0,Y 390.051,Z 391.901,A -85,B 0,C 180,E1 -11732.719,E2 -11732.719} C_VEL
LIN {X 0,Y 390.063,Z 391.895,A -85,B 0,C 180,E1 -11735.823,E2 -11735.823} C_VEL
LIN {X 0,Y 390.051,Z 391.897,A -85,B 0,C 180,E1 -11739.211,E2 -11739.211} C_VEL
LIN {X 0,Y 390.044,Z 391.901,A -85,B 0,C 180,E1 -11742.371,E2 -11742.371} C_VEL
LIN {X 0,Y 390.049,Z 391.897,A -85,B 0,C 180,E1 -11745.352,E2 -11745.352} C_VEL
LIN {X 0,Y 390.032,Z 391.902,A -85,B 0,C 180,E1 -11748.183,E2 -11748.183} C_VEL
LIN {X 0,Y 390.087,Z 391.895,A -85,B 0,C 180,E1 -11750.904,E2 -11750.904} C_VEL
LIN {X 0,Y 390.089,Z 391.895,A -85,B 0,C 180,E1 -11754.79,E2 -11754.79} C_VEL
LIN {X 0,Y 390.027,Z 391.904,A -85,B 0,C 180,E1 -11758.493,E2 -11758.493} C_VEL
LIN {X 0,Y 390.12,Z 391.891,A -85,B 0,C 180,E1 -11762.067,E2 -11762.067} C_VEL
LIN {X 0,Y 390.081,Z 391.893,A -85,B 0,C 180,E1 -11765.516,E2 -11765.516} C_VEL
LIN {X 0,Y 390.056,Z 391.897,A -85,B 0,C 180,E1 -11768.874,E2 -11768.874} C_VEL
LIN {X 0,Y 390.127,Z 391.891,A -85,B 0,C 180,E1 -11772.163,E2 -11772.163} C_VEL
LIN {X 0,Y 390.142,Z 391.886,A -85,B 0,C 180,E1 -11775.389,E2 -11775.389} C_VEL
LIN {X 0,Y 390.146,Z 391.888,A -85,B 0,C 180,E1 -11778.568,E2 -11778.568} C_VEL
LIN {X 0,Y 390.303,Z 391.869,A -85,B 0,C 180,E1 -11782.028,E2 -11782.028} C_VEL
LIN {X 0,Y 390.219,Z 391.876,A -85,B 0,C 180,E1 -11784.83,E2 -11784.83} C_VEL
LIN {X 0,Y 390.412,Z 391.855,A -85,B 0,C 180,E1 -11787.933,E2 -11787.933} C_VEL
LIN {X 0,Y 390.541,Z 391.84,A -85,B 0,C 180,E1 -11789.996,E2 -11789.996} C_VEL
LIN {X 0,Y 390.306,Z 391.865,A -85,B 0,C 180,E1 -11793.093,E2 -11793.093} C_VEL
LIN {X 0,Y 390.321,Z 391.867,A -85,B 0,C 180,E1 -11796.198,E2 -11796.198} C_VEL
LIN {X 0,Y 390.304,Z 391.869,A -85,B 0,C 180,E1 -11798.278,E2 -11798.278} C_VEL
LIN {X 0,Y 390.165,Z 391.885,A -85,B 0,C 180,E1 -11802.479,E2 -11802.479} C_VEL
LIN {X 0,Y 390.13,Z 391.889,A -85,B 0,C 180,E1 -11805.673,E2 -11805.673} C_VEL
LIN {X 0,Y 390.089,Z 391.892,A -85,B 0,C 180,E1 -11808.918,E2 -11808.918} C_VEL
LIN {X 0,Y 390.022,Z 391.904,A -85,B 0,C 180,E1 -11812.23,E2 -11812.23} C_VEL
LIN {X 0,Y 390.036,Z 391.9,A -85,B 0,C 180,E1 -11814.479,E2 -11814.479} C_VEL
LIN {X 0,Y 389.987,Z 391.905,A -85,B 0,C 180,E1 -11816.772,E2 -11816.772} C_VEL
LIN {X 0,Y 389.582,Z 391.961,A -85,B 0,C 180,E1 -11820.334,E2 -11820.334} C_VEL
LIN {X 0,Y 389.495,Z 391.97,A -85,B 0,C 180,E1 -11820.777,E2 -11820.777} C_VEL
LIN {X 0,Y 388.705,Z 392.163,A -85,B 0,C 180,E1 -11821.638,E2 -11821.638} C_VEL
LIN {X 0,Y 385.712,Z 393.076,A -85,B 0,C 180,E1 -11823.03,E2 -11823.03} C_VEL
LIN {X 0,Y 383.228,Z 394.131,A -85,B 0,C 180,E1 -11824.151,E2 -11824.151} C_VEL
LIN {X 0,Y 382.159,Z 394.994,A -85,B 0,C 180,E1 -11825.019,E2 -11825.019} C_VEL
LIN {X 0,Y 382.067,Z 395.278,A -85,B 0,C 180,E1 -11825.313,E2 -11825.313} C_VEL
LIN {X 0,Y 382.033,Z 398.594,A -85,B 0,C 180,E1 -11828.711,E2 -11828.711} C_VEL
LIN {X 0,Y 381.96,Z 401.357,A -85,B 0,C 180,E1 -11831.476,E2 -11831.476} C_VEL
LIN {X 0,Y 381.92,Z 403.533,A -85,B 0,C 180,E1 -11833.628,E2 -11833.628} C_VEL
LIN {X 0,Y 385.21,Z 417.244,A -85,B 0,C 180,E1 -11834.31,E2 -11834.31} C_VEL
LIN {X 0,Y 387.476,Z 428.272,A -85,B 0,C 180,E1 -11835.015,E2 -11835.015} C_VEL
LIN {X 0,Y 386.787,Z 440.597,A -85,B 0,C 180,E1 -11835.883,E2 -11835.883} C_VEL
LIN {X 0,Y 385.884,Z 452.542,A -85,B 0,C 180,E1 -11836.975,E2 -11836.975} C_VEL
LIN {X 0,Y 385.066,Z 463.232,A -85,B 0,C 180,E1 -11838.2,E2 -11838.2} C_VEL
LIN {X 0,Y 384.345,Z 472.548,A -85,B 0,C 180,E1 -11839.525,E2 -11839.525} C_VEL
LIN {X 0,Y 383.522,Z 481.676,A -85,B 0,C 180,E1 -11841.126,E2 -11841.126} C_VEL
LIN {X 0,Y 382.94,Z 488.993,A -85,B 0,C 180,E1 -11842.726,E2 -11842.726} C_VEL
LIN {X 0,Y 382.421,Z 495.746,A -85,B 0,C 180,E1 -11844.628,E2 -11844.628} C_VEL
LIN {X 0,Y 382.065,Z 500.781,A -85,B 0,C 180,E1 -11846.508,E2 -11846.508} C_VEL
LIN {X 0,Y 381.876,Z 503.384,A -85,B 0,C 180,E1 -11847.831,E2 -11847.831} C_VEL
LIN {X 0,Y 381.698,Z 505.119,A -85,B 0,C 180,E1 -11848.967,E2 -11848.967} C_VEL
LIN {X 0,Y 381.62,Z 506.381,A -85,B 0,C 180,E1 -11850.184,E2 -11850.184} C_VEL
LIN {X 0,Y 381.6,Z 507.324,A -85,B 0,C 180,E1 -11852.12,E2 -11852.12} C_VEL
LIN {X 0,Y 381.633,Z 507.052,A -85,B 0,C 180,E1 -11853.771,E2 -11853.771} C_VEL
LIN {X 0,Y 381.766,Z 506.268,A -85,B 0,C 180,E1 -11854.951,E2 -11854.951} C_VEL
LIN {X 0,Y 382.048,Z 503.84,A -85,B 0,C 180,E1 -11856.88,E2 -11856.88} C_VEL
LIN {X 0,Y 382.387,Z 500.855,A -85,B 0,C 180,E1 -11858.434,E2 -11858.434} C_VEL
LIN {X 0,Y 382.823,Z 496.391,A -85,B 0,C 180,E1 -11860.147,E2 -11860.147} C_VEL
LIN {X 0,Y 383.392,Z 490.624,A -85,B 0,C 180,E1 -11861.844,E2 -11861.844} C_VEL
LIN {X 0,Y 384.232,Z 483.282,A -85,B 0,C 180,E1 -11863.531,E2 -11863.531} C_VEL
LIN {X 0,Y 385.222,Z 474.115,A -85,B 0,C 180,E1 -11865.203,E2 -11865.203} C_VEL
LIN {X 0,Y 386.233,Z 464.638,A -85,B 0,C 180,E1 -11866.586,E2 -11866.586} C_VEL
LIN {X 0,Y 387.22,Z 454.421,A -85,B 0,C 180,E1 -11867.788,E2 -11867.788} C_VEL
LIN {X 0,Y 388.159,Z 443.511,A -85,B 0,C 180,E1 -11868.824,E2 -11868.824} C_VEL
LIN {X 0,Y 389.08,Z 431.154,A -85,B 0,C 180,E1 -11869.739,E2 -11869.739} C_VEL
LIN {X 0,Y 387.495,Z 422.996,A -85,B 0,C 180,E1 -11870.345,E2 -11870.345} C_VEL
LIN {X 0,Y 383.658,Z 410.293,A -85,B 0,C 180,E1 -11871.204,E2 -11871.204} C_VEL
LIN {X 0,Y 382.411,Z 406.195,A -85,B 0,C 180,E1 -11871.481,E2 -11871.481} C_VEL
LIN {X 0,Y 382.696,Z 403.435,A -85,B 0,C 180,E1 -11874.733,E2 -11874.733} C_VEL
LIN {X 0,Y 383.024,Z 399.206,A -85,B 0,C 180,E1 -11880.001,E2 -11880.001} C_VEL
LIN {X 0,Y 383.077,Z 397.63,A -85,B 0,C 180,E1 -11882.104,E2 -11882.104} C_VEL
LIN {X 0,Y 383.352,Z 394.591,A -85,B 0,C 180,E1 -11886.316,E2 -11886.316} C_VEL
LIN {X 0,Y 383.242,Z 393.213,A -85,B 0,C 180,E1 -11888.437,E2 -11888.437} C_VEL
LIN {X 0,Y 383.125,Z 392.764,A -85,B 0,C 180,E1 -11889.504,E2 -11889.504} C_VEL
LIN {X 0,Y 383.109,Z 392.766,A -85,B 0,C 180,E1 -11892.718,E2 -11892.718} C_VEL
LIN {X 0,Y 383.066,Z 392.771,A -85,B 0,C 180,E1 -11895.975,E2 -11895.975} C_VEL
LIN {X 0,Y 383.047,Z 392.773,A -85,B 0,C 180,E1 -11899.285,E2 -11899.285} C_VEL
LIN {X 0,Y 383.026,Z 392.773,A -85,B 0,C 180,E1 -11902.665,E2 -11902.665} C_VEL
LIN {X 0,Y 383.05,Z 392.77,A -85,B 0,C 180,E1 -11906.126,E2 -11906.126} C_VEL
LIN {X 0,Y 383.02,Z 392.776,A -85,B 0,C 180,E1 -11908.495,E2 -11908.495} C_VEL
LIN {X 0,Y 382.983,Z 392.78,A -85,B 0,C 180,E1 -11912.153,E2 -11912.153} C_VEL
LIN {X 0,Y 382.992,Z 392.78,A -85,B 0,C 180,E1 -11914.672,E2 -11914.672} C_VEL
LIN {X 0,Y 382.979,Z 392.782,A -85,B 0,C 180,E1 -11917.908,E2 -11917.908} C_VEL
LIN {X 0,Y 383.024,Z 392.776,A -85,B 0,C 180,E1 -11921.343,E2 -11921.343} C_VEL
LIN {X 0,Y 383.251,Z 393.887,A -85,B 0,C 180,E1 -11922.826,E2 -11922.826} C_VEL
LIN {X 0,Y 383.815,Z 397.152,A -85,B 0,C 180,E1 -11925.915,E2 -11925.915} C_VEL
LIN {X 0,Y 384.446,Z 400.813,A -85,B 0,C 180,E1 -11928.851,E2 -11928.851} C_VEL
LIN {X 0,Y 385.288,Z 405.819,A -85,B 0,C 180,E1 -11932.357,E2 -11932.357} C_VEL
LIN {X 0,Y 385.392,Z 408.962,A -85,B 0,C 180,E1 -11934.305,E2 -11934.305} C_VEL
LIN {X 0,Y 384.676,Z 414.13,A -85,B 0,C 180,E1 -11937.185,E2 -11937.185} C_VEL
LIN {X 0,Y 383.723,Z 421.415,A -85,B 0,C 180,E1 -11940.97,E2 -11940.97} C_VEL
LIN {X 0,Y 383.254,Z 427.516,A -85,B 0,C 180,E1 -11943.969,E2 -11943.969} C_VEL
LIN {X 0,Y 382.651,Z 435.907,A -85,B 0,C 180,E1 -11947.887,E2 -11947.887} C_VEL
LIN {X 0,Y 382.35,Z 441.926,A -85,B 0,C 180,E1 -11950.527,E2 -11950.527} C_VEL
LIN {X 0,Y 385.189,Z 456.15,A -85,B 0,C 180,E1 -11951.239,E2 -11951.239} C_VEL
LIN {X 0,Y 386.673,Z 468.566,A -85,B 0,C 180,E1 -11952.007,E2 -11952.007} C_VEL
LIN {X 0,Y 387.254,Z 479.964,A -85,B 0,C 180,E1 -11952.852,E2 -11952.852} C_VEL
LIN {X 0,Y 386.166,Z 492.07,A -85,B 0,C 180,E1 -11953.891,E2 -11953.891} C_VEL
LIN {X 0,Y 385.06,Z 502.896,A -85,B 0,C 180,E1 -11955.065,E2 -11955.065} C_VEL
LIN {X 0,Y 384.153,Z 511.841,A -85,B 0,C 180,E1 -11956.246,E2 -11956.246} C_VEL
LIN {X 0,Y 383.489,Z 520.15,A -85,B 0,C 180,E1 -11957.569,E2 -11957.569} C_VEL
LIN {X 0,Y 382.653,Z 528.352,A -85,B 0,C 180,E1 -11959.153,E2 -11959.153} C_VEL
LIN {X 0,Y 382.244,Z 533.95,A -85,B 0,C 180,E1 -11960.479,E2 -11960.479} C_VEL
LIN {X 0,Y 381.904,Z 539.464,A -85,B 0,C 180,E1 -11962.071,E2 -11962.071} C_VEL
LIN {X 0,Y 381.675,Z 544.367,A -85,B 0,C 180,E1 -11963.903,E2 -11963.903} C_VEL
LIN {X 0,Y 381.655,Z 547.9,A -85,B 0,C 180,E1 -11965.78,E2 -11965.78} C_VEL
LIN {X 0,Y 381.751,Z 550.295,A -85,B 0,C 180,E1 -11967.894,E2 -11967.894} C_VEL
LIN {X 0,Y 381.732,Z 550.856,A -85,B 0,C 180,E1 -11968.949,E2 -11968.949} C_VEL
LIN {X 0,Y 381.727,Z 550.983,A -85,B 0,C 180,E1 -11970.004,E2 -11970.004} C_VEL
LIN {X 0,Y 381.733,Z 550.711,A -85,B 0,C 180,E1 -11971.059,E2 -11971.059} C_VEL
LIN {X 0,Y 381.778,Z 550.042,A -85,B 0,C 180,E1 -11972.114,E2 -11972.114} C_VEL
LIN {X 0,Y 381.665,Z 548.92,A -85,B 0,C 180,E1 -11973.171,E2 -11973.171} C_VEL
LIN {X 0,Y 381.665,Z 547.357,A -85,B 0,C 180,E1 -11974.228,E2 -11974.228} C_VEL
LIN {X 0,Y 381.726,Z 545.369,A -85,B 0,C 180,E1 -11975.286,E2 -11975.286} C_VEL
LIN {X 0,Y 381.789,Z 541.475,A -85,B 0,C 180,E1 -11976.876,E2 -11976.876} C_VEL
LIN {X 0,Y 382.013,Z 536.425,A -85,B 0,C 180,E1 -11978.467,E2 -11978.467} C_VEL
LIN {X 0,Y 382.375,Z 530.059,A -85,B 0,C 180,E1 -11980.059,E2 -11980.059} C_VEL
LIN {X 0,Y 382.979,Z 522.079,A -85,B 0,C 180,E1 -11981.649,E2 -11981.649} C_VEL
LIN {X 0,Y 383.621,Z 513.958,A -85,B 0,C 180,E1 -11982.972,E2 -11982.972} C_VEL
LIN {X 0,Y 384.312,Z 504.447,A -85,B 0,C 180,E1 -11984.25,E2 -11984.25} C_VEL
LIN {X 0,Y 385.145,Z 494.437,A -85,B 0,C 180,E1 -11985.346,E2 -11985.346} C_VEL
LIN {X 0,Y 386.17,Z 482.404,A -85,B 0,C 180,E1 -11986.388,E2 -11986.388} C_VEL
LIN {X 0,Y 386.31,Z 476.949,A -85,B 0,C 180,E1 -11986.79,E2 -11986.79} C_VEL
LIN {X 0,Y 384.999,Z 463.809,A -85,B 0,C 180,E1 -11987.64,E2 -11987.64} C_VEL
LIN {X 0,Y 383.267,Z 451.217,A -85,B 0,C 180,E1 -11988.253,E2 -11988.253} C_VEL
LIN {X 0,Y 382.221,Z 444.201,A -85,B 0,C 180,E1 -11988.531,E2 -11988.531} C_VEL
LIN {X 0,Y 382.658,Z 436.172,A -85,B 0,C 180,E1 -11992.121,E2 -11992.121} C_VEL
LIN {X 0,Y 383.135,Z 428.773,A -85,B 0,C 180,E1 -11995.495,E2 -11995.495} C_VEL
LIN {X 0,Y 383.784,Z 421.167,A -85,B 0,C 180,E1 -11999.034,E2 -11999.034} C_VEL
LIN {X 0,Y 384.399,Z 414.906,A -85,B 0,C 180,E1 -12002.023,E2 -12002.023} C_VEL
LIN {X 0,Y 385.066,Z 409.268,A -85,B 0,C 180,E1 -12004.782,E2 -12004.782} C_VEL
LIN {X 0,Y 385.096,Z 404.85,A -85,B 0,C 180,E1 -12007.035,E2 -12007.035} C_VEL
LIN {X 0,Y 384.054,Z 398.493,A -85,B 0,C 180,E1 -12010.517,E2 -12010.517} C_VEL
LIN {X 0,Y 383.038,Z 392.771,A -85,B 0,C 180,E1 -12013.838,E2 -12013.838} C_VEL
LIN {X 0,Y 383.026,Z 392.777,A -85,B 0,C 180,E1 -12017.241,E2 -12017.241} C_VEL
LIN {X 0,Y 383,Z 392.775,A -85,B 0,C 180,E1 -12020.42,E2 -12020.42} C_VEL
LIN {X 0,Y 383.029,Z 392.772,A -85,B 0,C 180,E1 -12024.044,E2 -12024.044} C_VEL
LIN {X 0,Y 383,Z 392.778,A -85,B 0,C 180,E1 -12027.579,E2 -12027.579} C_VEL
LIN {X 0,Y 382.994,Z 392.776,A -85,B 0,C 180,E1 -12030.299,E2 -12030.299} C_VEL
LIN {X 0,Y 383.019,Z 392.772,A -85,B 0,C 180,E1 -12034.045,E2 -12034.045} C_VEL
LIN {X 0,Y 383.005,Z 392.777,A -85,B 0,C 180,E1 -12037.334,E2 -12037.334} C_VEL
LIN {X 0,Y 383.073,Z 392.769,A -85,B 0,C 180,E1 -12040.716,E2 -12040.716} C_VEL
LIN {X 0,Y 383.093,Z 392.764,A -85,B 0,C 180,E1 -12044.026,E2 -12044.026} C_VEL
LIN {X 0,Y 383.15,Z 392.76,A -85,B 0,C 180,E1 -12047.283,E2 -12047.283} C_VEL
LIN {X 0,Y 383.156,Z 392.757,A -85,B 0,C 180,E1 -12050.497,E2 -12050.497} C_VEL
LIN {X 0,Y 383.274,Z 392.741,A -85,B 0,C 180,E1 -12053.683,E2 -12053.683} C_VEL
LIN {X 0,Y 383.396,Z 392.726,A -85,B 0,C 180,E1 -12057.898,E2 -12057.898} C_VEL
LIN {X 0,Y 383.525,Z 392.71,A -85,B 0,C 180,E1 -12059.999,E2 -12059.999} C_VEL
LIN {X 0,Y 383.224,Z 392.75,A -85,B 0,C 180,E1 -12063.153,E2 -12063.153} C_VEL
LIN {X 0,Y 383.233,Z 392.746,A -85,B 0,C 180,E1 -12066.53,E2 -12066.53} C_VEL
LIN {X 0,Y 383.154,Z 392.757,A -85,B 0,C 180,E1 -12069.501,E2 -12069.501} C_VEL
LIN {X 0,Y 383.138,Z 392.758,A -85,B 0,C 180,E1 -12073.534,E2 -12073.534} C_VEL
LIN {X 0,Y 383.105,Z 392.766,A -85,B 0,C 180,E1 -12077.068,E2 -12077.068} C_VEL
LIN {X 0,Y 383.039,Z 392.775,A -85,B 0,C 180,E1 -12080.645,E2 -12080.645} C_VEL
LIN {X 0,Y 383.032,Z 392.771,A -85,B 0,C 180,E1 -12083.806,E2 -12083.806} C_VEL
LIN {X 0,Y 383.089,Z 392.766,A -85,B 0,C 180,E1 -12086.121,E2 -12086.121} C_VEL
LIN {X 0,Y 382.997,Z 392.776,A -85,B 0,C 180,E1 -12089.698,E2 -12089.698} C_VEL
LIN {X 0,Y 383.011,Z 392.774,A -85,B 0,C 180,E1 -12093.399,E2 -12093.399} C_VEL
LIN {X 0,Y 383.039,Z 392.772,A -85,B 0,C 180,E1 -12096.162,E2 -12096.162} C_VEL
LIN {X 0,Y 383.007,Z 392.775,A -85,B 0,C 180,E1 -12099.957,E2 -12099.957} C_VEL
LIN {X 0,Y 383.012,Z 392.777,A -85,B 0,C 180,E1 -12102.776,E2 -12102.776} C_VEL
LIN {X 0,Y 383.002,Z 392.775,A -85,B 0,C 180,E1 -12105.786,E2 -12105.786} C_VEL
LIN {X 0,Y 382.987,Z 392.78,A -85,B 0,C 180,E1 -12108.794,E2 -12108.794} C_VEL
LIN {X 0,Y 383.002,Z 392.777,A -85,B 0,C 180,E1 -12112.094,E2 -12112.094} C_VEL
LIN {X 0,Y 383.022,Z 392.772,A -85,B 0,C 180,E1 -12115.329,E2 -12115.329} C_VEL
LIN {X 0,Y 382.986,Z 392.778,A -85,B 0,C 180,E1 -12119.078,E2 -12119.078} C_VEL
LIN {X 0,Y 383.059,Z 392.771,A -85,B 0,C 180,E1 -12122.695,E2 -12122.695} C_VEL
LIN {X 0,Y 383.054,Z 392.769,A -85,B 0,C 180,E1 -12125.036,E2 -12125.036} C_VEL
LIN {X 0,Y 382.994,Z 392.78,A -85,B 0,C 180,E1 -12128.466,E2 -12128.466} C_VEL
LIN {X 0,Y 383.062,Z 392.769,A -85,B 0,C 180,E1 -12131.823,E2 -12131.823} C_VEL
LIN {X 0,Y 383.108,Z 392.762,A -85,B 0,C 180,E1 -12135.115,E2 -12135.115} C_VEL
LIN {X 0,Y 383.095,Z 392.767,A -85,B 0,C 180,E1 -12138.354,E2 -12138.354} C_VEL
LIN {X 0,Y 383.259,Z 392.746,A -85,B 0,C 180,E1 -12141.972,E2 -12141.972} C_VEL
LIN {X 0,Y 383.191,Z 392.752,A -85,B 0,C 180,E1 -12144.735,E2 -12144.735} C_VEL
LIN {X 0,Y 383.379,Z 392.732,A -85,B 0,C 180,E1 -12147.895,E2 -12147.895} C_VEL
LIN {X 0,Y 383.51,Z 392.715,A -85,B 0,C 180,E1 -12149.996,E2 -12149.996} C_VEL
LIN {X 0,Y 383.242,Z 392.745,A -85,B 0,C 180,E1 -12153.15,E2 -12153.15} C_VEL
LIN {X 0,Y 383.278,Z 392.745,A -85,B 0,C 180,E1 -12156.312,E2 -12156.312} C_VEL
LIN {X 0,Y 383.249,Z 392.747,A -85,B 0,C 180,E1 -12158.432,E2 -12158.432} C_VEL
LIN {X 0,Y 383.095,Z 392.765,A -85,B 0,C 180,E1 -12161.638,E2 -12161.638} C_VEL
LIN {X 0,Y 383.1,Z 392.763,A -85,B 0,C 180,E1 -12164.878,E2 -12164.878} C_VEL
LIN {X 0,Y 383.073,Z 392.77,A -85,B 0,C 180,E1 -12168.168,E2 -12168.168} C_VEL
LIN {X 0,Y 382.975,Z 392.78,A -85,B 0,C 180,E1 -12171.527,E2 -12171.527} C_VEL
LIN {X 0,Y 382.998,Z 392.775,A -85,B 0,C 180,E1 -12174.959,E2 -12174.959} C_VEL
LIN {X 0,Y 382.788,Z 392.806,A -85,B 0,C 180,E1 -12178.205,E2 -12178.205} C_VEL
LIN {X 0,Y 382.425,Z 392.85,A -85,B 0,C 180,E1 -12180.963,E2 -12180.963} C_VEL
LIN {X 0,Y 382.254,Z 392.873,A -85,B 0,C 180,E1 -12182.251,E2 -12182.251} C_VEL
LIN {X 0,Y 382.128,Z 394.165,A -85,B 0,C 180,E1 -12184.146,E2 -12184.146} C_VEL
LIN {X 0,Y 382.067,Z 395.278,A -85,B 0,C 180,E1 -12185.313,E2 -12185.313} C_VEL
LIN {X 0,Y 381.387,Z 396.185,A -85,B 0,C 180,E1 -12186.183,E2 -12186.183} C_VEL
LIN {X 0,Y 378.525,Z 397.852,A -85,B 0,C 180,E1 -12187.592,E2 -12187.592} C_VEL
LIN {X 0,Y 376.09,Z 399.203,A -85,B 0,C 180,E1 -12188.73,E2 -12188.73} C_VEL
LIN {X 0,Y 375.019,Z 400.168,A -85,B 0,C 180,E1 -12189.612,E2 -12189.612} C_VEL
LIN {X 0,Y 374.918,Z 400.472,A -85,B 0,C 180,E1 -12189.912,E2 -12189.912} C_VEL
LIN {X 0,Y 374.862,Z 403.873,A -85,B 0,C 180,E1 -12193.313,E2 -12193.313} C_VEL
LIN {X 0,Y 378.568,Z 419.495,A -85,B 0,C 180,E1 -12194.141,E2 -12194.141} C_VEL
LIN {X 0,Y 380.533,Z 428.839,A -85,B 0,C 180,E1 -12194.77,E2 -12194.77} C_VEL
LIN {X 0,Y 379.912,Z 440.53,A -85,B 0,C 180,E1 -12195.609,E2 -12195.609} C_VEL
LIN {X 0,Y 379.042,Z 452.211,A -85,B 0,C 180,E1 -12196.685,E2 -12196.685} C_VEL
LIN {X 0,Y 378.114,Z 463.592,A -85,B 0,C 180,E1 -12198.002,E2 -12198.002} C_VEL
LIN {X 0,Y 377.384,Z 472.752,A -85,B 0,C 180,E1 -12199.324,E2 -12199.324} C_VEL
LIN {X 0,Y 376.53,Z 481.679,A -85,B 0,C 180,E1 -12200.908,E2 -12200.908} C_VEL
LIN {X 0,Y 375.902,Z 489.268,A -85,B 0,C 180,E1 -12202.583,E2 -12202.583} C_VEL
LIN {X 0,Y 375.459,Z 494.561,A -85,B 0,C 180,E1 -12204.039,E2 -12204.039} C_VEL
LIN {X 0,Y 375.105,Z 499.618,A -85,B 0,C 180,E1 -12205.801,E2 -12205.801} C_VEL
LIN {X 0,Y 374.85,Z 503.294,A -85,B 0,C 180,E1 -12207.522,E2 -12207.522} C_VEL
LIN {X 0,Y 374.571,Z 506.298,A -85,B 0,C 180,E1 -12209.654,E2 -12209.654} C_VEL
LIN {X 0,Y 374.518,Z 507.237,A -85,B 0,C 180,E1 -12210.799,E2 -12210.799} C_VEL
LIN {X 0,Y 374.514,Z 507.71,A -85,B 0,C 180,E1 -12212.023,E2 -12212.023} C_VEL
LIN {X 0,Y 374.533,Z 507.709,A -85,B 0,C 180,E1 -12213.235,E2 -12213.235} C_VEL
LIN {X 0,Y 374.611,Z 507.15,A -85,B 0,C 180,E1 -12214.439,E2 -12214.439} C_VEL
LIN {X 0,Y 374.773,Z 506.123,A -85,B 0,C 180,E1 -12215.635,E2 -12215.635} C_VEL
LIN {X 0,Y 375.114,Z 503.64,A -85,B 0,C 180,E1 -12217.415,E2 -12217.415} C_VEL
LIN {X 0,Y 375.532,Z 499.593,A -85,B 0,C 180,E1 -12219.332,E2 -12219.332} C_VEL
LIN {X 0,Y 376.005,Z 495.138,A -85,B 0,C 180,E1 -12220.908,E2 -12220.908} C_VEL
LIN {X 0,Y 376.761,Z 488.88,A -85,B 0,C 180,E1 -12222.636,E2 -12222.636} C_VEL
LIN {X 0,Y 377.686,Z 481.055,A -85,B 0,C 180,E1 -12224.348,E2 -12224.348} C_VEL
LIN {X 0,Y 378.625,Z 472.747,A -85,B 0,C 180,E1 -12225.799,E2 -12225.799} C_VEL
LIN {X 0,Y 379.628,Z 463.154,A -85,B 0,C 180,E1 -12227.165,E2 -12227.165} C_VEL
LIN {X 0,Y 380.798,Z 452.159,A -85,B 0,C 180,E1 -12228.423,E2 -12228.423} C_VEL
LIN {X 0,Y 381.855,Z 439.786,A -85,B 0,C 180,E1 -12229.531,E2 -12229.531} C_VEL
LIN {X 0,Y 382.438,Z 432.204,A -85,B 0,C 180,E1 -12230.084,E2 -12230.084} C_VEL
LIN {X 0,Y 380.457,Z 422.857,A -85,B 0,C 180,E1 -12230.818,E2 -12230.818} C_VEL
LIN {X 0,Y 376.603,Z 410.53,A -85,B 0,C 180,E1 -12231.681,E2 -12231.681} C_VEL
LIN {X 0,Y 375.393,Z 406.719,A -85,B 0,C 180,E1 -12231.93,E2 -12231.93} C_VEL
LIN {X 0,Y 375.655,Z 404.471,A -85,B 0,C 180,E1 -12234.634,E2 -12234.634} C_VEL
LIN {X 0,Y 376.001,Z 400.244,A -85,B 0,C 180,E1 -12240.001,E2 -12240.001} C_VEL
LIN {X 0,Y 376.065,Z 398.681,A -85,B 0,C 180,E1 -12242.143,E2 -12242.143} C_VEL
LIN {X 0,Y 376.343,Z 395.69,A -85,B 0,C 180,E1 -12246.434,E2 -12246.434} C_VEL
LIN {X 0,Y 376.224,Z 394.315,A -85,B 0,C 180,E1 -12248.596,E2 -12248.596} C_VEL
LIN {X 0,Y 376.093,Z 393.685,A -85,B 0,C 180,E1 -12249.683,E2 -12249.683} C_VEL
LIN {X 0,Y 376.056,Z 393.644,A -85,B 0,C 180,E1 -12253.66,E2 -12253.66} C_VEL
LIN {X 0,Y 376.035,Z 393.647,A -85,B 0,C 180,E1 -12257.622,E2 -12257.622} C_VEL
LIN {X 0,Y 376.009,Z 393.648,A -85,B 0,C 180,E1 -12260.86,E2 -12260.86} C_VEL
LIN {X 0,Y 375.971,Z 393.652,A -85,B 0,C 180,E1 -12264.284,E2 -12264.284} C_VEL
LIN {X 0,Y 375.99,Z 393.651,A -85,B 0,C 180,E1 -12266.655,E2 -12266.655} C_VEL
LIN {X 0,Y 375.947,Z 393.655,A -85,B 0,C 180,E1 -12269.082,E2 -12269.082} C_VEL
LIN {X 0,Y 375.922,Z 393.658,A -85,B 0,C 180,E1 -12272.832,E2 -12272.832} C_VEL
LIN {X 0,Y 375.932,Z 393.658,A -85,B 0,C 180,E1 -12275.419,E2 -12275.419} C_VEL
LIN {X 0,Y 375.954,Z 393.656,A -85,B 0,C 180,E1 -12278.275,E2 -12278.275} C_VEL
LIN {X 0,Y 375.977,Z 393.768,A -85,B 0,C 180,E1 -12280.863,E2 -12280.863} C_VEL
LIN {X 0,Y 376.476,Z 396.339,A -85,B 0,C 180,E1 -12283.687,E2 -12283.687} C_VEL
LIN {X 0,Y 377.017,Z 399.546,A -85,B 0,C 180,E1 -12286.637,E2 -12286.637} C_VEL
LIN {X 0,Y 377.68,Z 403.447,A -85,B 0,C 180,E1 -12289.725,E2 -12289.725} C_VEL
LIN {X 0,Y 378.276,Z 406.928,A -85,B 0,C 180,E1 -12292.192,E2 -12292.192} C_VEL
LIN {X 0,Y 378.404,Z 410.09,A -85,B 0,C 180,E1 -12294.2,E2 -12294.2} C_VEL
LIN {X 0,Y 377.604,Z 415.581,A -85,B 0,C 180,E1 -12297.339,E2 -12297.339} C_VEL
LIN {X 0,Y 376.65,Z 423.03,A -85,B 0,C 180,E1 -12301.282,E2 -12301.282} C_VEL
LIN {X 0,Y 376.071,Z 429.584,A -85,B 0,C 180,E1 -12304.549,E2 -12304.549} C_VEL
LIN {X 0,Y 375.558,Z 436.882,A -85,B 0,C 180,E1 -12308.026,E2 -12308.026} C_VEL
LIN {X 0,Y 375.317,Z 441.224,A -85,B 0,C 180,E1 -12310.027,E2 -12310.027} C_VEL
LIN {X 0,Y 378.248,Z 455.739,A -85,B 0,C 180,E1 -12310.802,E2 -12310.802} C_VEL
LIN {X 0,Y 379.851,Z 468.357,A -85,B 0,C 180,E1 -12311.62,E2 -12311.62} C_VEL
LIN {X 0,Y 380.452,Z 480.316,A -85,B 0,C 180,E1 -12312.536,E2 -12312.536} C_VEL
LIN {X 0,Y 379.341,Z 492.234,A -85,B 0,C 180,E1 -12313.593,E2 -12313.593} C_VEL
LIN {X 0,Y 378.091,Z 504.006,A -85,B 0,C 180,E1 -12314.921,E2 -12314.921} C_VEL
LIN {X 0,Y 377.122,Z 513.586,A -85,B 0,C 180,E1 -12316.259,E2 -12316.259} C_VEL
LIN {X 0,Y 376.37,Z 521.511,A -85,B 0,C 180,E1 -12317.604,E2 -12317.604} C_VEL
LIN {X 0,Y 375.528,Z 529.313,A -85,B 0,C 180,E1 -12319.218,E2 -12319.218} C_VEL
LIN {X 0,Y 375.072,Z 535.657,A -85,B 0,C 180,E1 -12320.84,E2 -12320.84} C_VEL
LIN {X 0,Y 374.763,Z 540.725,A -85,B 0,C 180,E1 -12322.461,E2 -12322.461} C_VEL
LIN {X 0,Y 374.591,Z 544.331,A -85,B 0,C 180,E1 -12323.926,E2 -12323.926} C_VEL
LIN {X 0,Y 374.579,Z 547.547,A -85,B 0,C 180,E1 -12325.7,E2 -12325.7} C_VEL
LIN {X 0,Y 374.65,Z 549.915,A -85,B 0,C 180,E1 -12327.854,E2 -12327.854} C_VEL
LIN {X 0,Y 374.663,Z 550.448,A -85,B 0,C 180,E1 -12328.929,E2 -12328.929} C_VEL
LIN {X 0,Y 374.656,Z 550.561,A -85,B 0,C 180,E1 -12330.004,E2 -12330.004} C_VEL
LIN {X 0,Y 374.665,Z 550.276,A -85,B 0,C 180,E1 -12331.079,E2 -12331.079} C_VEL
LIN {X 0,Y 374.691,Z 549.592,A -85,B 0,C 180,E1 -12332.154,E2 -12332.154} C_VEL
LIN {X 0,Y 374.572,Z 548.44,A -85,B 0,C 180,E1 -12333.231,E2 -12333.231} C_VEL
LIN {X 0,Y 374.602,Z 545.929,A -85,B 0,C 180,E1 -12334.847,E2 -12334.847} C_VEL
LIN {X 0,Y 374.671,Z 542.369,A -85,B 0,C 180,E1 -12336.466,E2 -12336.466} C_VEL
LIN {X 0,Y 374.854,Z 537.67,A -85,B 0,C 180,E1 -12338.087,E2 -12338.087} C_VEL
LIN {X 0,Y 375.257,Z 530.566,A -85,B 0,C 180,E1 -12339.98,E2 -12339.98} C_VEL
LIN {X 0,Y 375.861,Z 522.864,A -85,B 0,C 180,E1 -12341.6,E2 -12341.6} C_VEL
LIN {X 0,Y 376.496,Z 514.975,A -85,B 0,C 180,E1 -12342.948,E2 -12342.948} C_VEL
LIN {X 0,Y 377.265,Z 504.765,A -85,B 0,C 180,E1 -12344.371,E2 -12344.371} C_VEL
LIN {X 0,Y 378.275,Z 493.486,A -85,B 0,C 180,E1 -12345.632,E2 -12345.632} C_VEL
LIN {X 0,Y 379.302,Z 481.294,A -85,B 0,C 180,E1 -12346.694,E2 -12346.694} C_VEL
LIN {X 0,Y 379.027,Z 473.707,A -85,B 0,C 180,E1 -12347.262,E2 -12347.262} C_VEL
LIN {X 0,Y 377.546,Z 460.502,A -85,B 0,C 180,E1 -12348.075,E2 -12348.075} C_VEL
LIN {X 0,Y 375.532,Z 446.545,A -85,B 0,C 180,E1 -12348.717,E2 -12348.717} C_VEL
LIN {X 0,Y 375.186,Z 443.881,A -85,B 0,C 180,E1 -12348.82,E2 -12348.82} C_VEL
LIN {X 0,Y 375.643,Z 435.731,A -85,B 0,C 180,E1 -12352.557,E2 -12352.557} C_VEL
LIN {X 0,Y 376.205,Z 427.763,A -85,B 0,C 180,E1 -12356.271,E2 -12356.271} C_VEL
LIN {X 0,Y 376.948,Z 419.516,A -85,B 0,C 180,E1 -12360.229,E2 -12360.229} C_VEL
LIN {X 0,Y 377.614,Z 413.629,A -85,B 0,C 180,E1 -12363.12,E2 -12363.12} C_VEL
LIN {X 0,Y 378.156,Z 408.258,A -85,B 0,C 180,E1 -12365.836,E2 -12365.836} C_VEL
LIN {X 0,Y 377.855,Z 404.468,A -85,B 0,C 180,E1 -12367.868,E2 -12367.868} C_VEL
LIN {X 0,Y 376.999,Z 399.354,A -85,B 0,C 180,E1 -12370.731,E2 -12370.731} C_VEL
LIN {X 0,Y 375.998,Z 393.648,A -85,B 0,C 180,E1 -12374.144,E2 -12374.144} C_VEL
LIN {X 0,Y 375.94,Z 393.657,A -85,B 0,C 180,E1 -12377.7,E2 -12377.7} C_VEL
LIN {X 0,Y 375.949,Z 393.654,A -85,B 0,C 180,E1 -12380.535,E2 -12380.535} C_VEL
LIN {X 0,Y 375.973,Z 393.654,A -85,B 0,C 180,E1 -12383.498,E2 -12383.498} C_VEL
LIN {X 0,Y 375.972,Z 393.651,A -85,B 0,C 180,E1 -12385.889,E2 -12385.889} C_VEL
LIN {X 0,Y 375.977,Z 393.651,A -85,B 0,C 180,E1 -12389.688,E2 -12389.688} C_VEL
LIN {X 0,Y 375.948,Z 393.653,A -85,B 0,C 180,E1 -12392.137,E2 -12392.137} C_VEL
LIN {X 0,Y 375.985,Z 393.65,A -85,B 0,C 180,E1 -12395.717,E2 -12395.717} C_VEL
LIN {X 0,Y 375.995,Z 393.651,A -85,B 0,C 180,E1 -12399.197,E2 -12399.197} C_VEL
LIN {X 0,Y 376.047,Z 393.643,A -85,B 0,C 180,E1 -12402.6,E2 -12402.6} C_VEL
LIN {X 0,Y 376.105,Z 393.634,A -85,B 0,C 180,E1 -12406.342,E2 -12406.342} C_VEL
LIN {X 0,Y 376.126,Z 393.632,A -85,B 0,C 180,E1 -12410.318,E2 -12410.318} C_VEL
LIN {X 0,Y 376.233,Z 393.619,A -85,B 0,C 180,E1 -12413.564,E2 -12413.564} C_VEL
LIN {X 0,Y 376.362,Z 393.602,A -85,B 0,C 180,E1 -12417.859,E2 -12417.859} C_VEL
LIN {X 0,Y 376.495,Z 393.585,A -85,B 0,C 180,E1 -12419.999,E2 -12419.999} C_VEL
LIN {X 0,Y 376.356,Z 393.603,A -85,B 0,C 180,E1 -12422.139,E2 -12422.139} C_VEL
LIN {X 0,Y 376.203,Z 393.623,A -85,B 0,C 180,E1 -12426.515,E2 -12426.515} C_VEL
LIN {X 0,Y 376.124,Z 393.632,A -85,B 0,C 180,E1 -12429.68,E2 -12429.68} C_VEL
LIN {X 0,Y 376.102,Z 393.634,A -85,B 0,C 180,E1 -12433.656,E2 -12433.656} C_VEL
LIN {X 0,Y 376.043,Z 393.642,A -85,B 0,C 180,E1 -12437.398,E2 -12437.398} C_VEL
LIN {X 0,Y 375.99,Z 393.652,A -85,B 0,C 180,E1 -12440.83,E2 -12440.83} C_VEL
LIN {X 0,Y 375.997,Z 393.649,A -85,B 0,C 180,E1 -12444.28,E2 -12444.28} C_VEL
LIN {X 0,Y 376.029,Z 393.648,A -85,B 0,C 180,E1 -12446.65,E2 -12446.65} C_VEL
LIN {X 0,Y 375.972,Z 393.654,A -85,B 0,C 180,E1 -12450.311,E2 -12450.311} C_VEL
LIN {X 0,Y 375.968,Z 393.653,A -85,B 0,C 180,E1 -12454.109,E2 -12454.109} C_VEL
LIN {X 0,Y 375.96,Z 393.656,A -85,B 0,C 180,E1 -12456.739,E2 -12456.739} C_VEL
LIN {X 0,Y 375.987,Z 393.649,A -85,B 0,C 180,E1 -12459.966,E2 -12459.966} C_VEL
LIN {X 0,Y 375.935,Z 393.655,A -85,B 0,C 180,E1 -12463.764,E2 -12463.764} C_VEL
LIN {X 0,Y 375.94,Z 393.658,A -85,B 0,C 180,E1 -12466.808,E2 -12466.808} C_VEL
LIN {X 0,Y 375.958,Z 393.656,A -85,B 0,C 180,E1 -12470.533,E2 -12470.533} C_VEL
LIN {X 0,Y 375.968,Z 393.651,A -85,B 0,C 180,E1 -12473.493,E2 -12473.493} C_VEL
LIN {X 0,Y 375.964,Z 393.653,A -85,B 0,C 180,E1 -12475.885,E2 -12475.885} C_VEL
LIN {X 0,Y 375.967,Z 393.651,A -85,B 0,C 180,E1 -12479.684,E2 -12479.684} C_VEL
LIN {X 0,Y 376.022,Z 393.644,A -85,B 0,C 180,E1 -12483.345,E2 -12483.345} C_VEL
LIN {X 0,Y 375.998,Z 393.649,A -85,B 0,C 180,E1 -12486.885,E2 -12486.885} C_VEL
LIN {X 0,Y 375.998,Z 393.651,A -85,B 0,C 180,E1 -12490.336,E2 -12490.336} C_VEL
LIN {X 0,Y 376.027,Z 393.644,A -85,B 0,C 180,E1 -12493.715,E2 -12493.715} C_VEL
LIN {X 0,Y 376.101,Z 393.634,A -85,B 0,C 180,E1 -12497.038,E2 -12497.038} C_VEL
LIN {X 0,Y 376.116,Z 393.637,A -85,B 0,C 180,E1 -12500.315,E2 -12500.315} C_VEL
LIN {X 0,Y 376.234,Z 393.619,A -85,B 0,C 180,E1 -12503.561,E2 -12503.561} C_VEL
LIN {X 0,Y 376.345,Z 393.607,A -85,B 0,C 180,E1 -12507.856,E2 -12507.856} C_VEL
LIN {X 0,Y 376.479,Z 393.591,A -85,B 0,C 180,E1 -12509.996,E2 -12509.996} C_VEL
LIN {X 0,Y 376.18,Z 393.624,A -85,B 0,C 180,E1 -12513.209,E2 -12513.209} C_VEL
LIN {X 0,Y 376.237,Z 393.62,A -85,B 0,C 180,E1 -12516.431,E2 -12516.431} C_VEL
LIN {X 0,Y 376.195,Z 393.624,A -85,B 0,C 180,E1 -12518.591,E2 -12518.591} C_VEL
LIN {X 0,Y 376.047,Z 393.644,A -85,B 0,C 180,E1 -12521.859,E2 -12521.859} C_VEL
LIN {X 0,Y 376.048,Z 393.641,A -85,B 0,C 180,E1 -12525.163,E2 -12525.163} C_VEL
LIN {X 0,Y 376.008,Z 393.648,A -85,B 0,C 180,E1 -12528.522,E2 -12528.522} C_VEL
LIN {X 0,Y 375.945,Z 393.658,A -85,B 0,C 180,E1 -12531.95,E2 -12531.95} C_VEL
LIN {X 0,Y 375.958,Z 393.655,A -85,B 0,C 180,E1 -12534.279,E2 -12534.279} C_VEL
LIN {X 0,Y 375.857,Z 393.665,A -85,B 0,C 180,E1 -12536.659,E2 -12536.659} C_VEL
LIN {X 0,Y 375.623,Z 393.695,A -85,B 0,C 180,E1 -12539.103,E2 -12539.103} C_VEL
LIN {X 0,Y 375.269,Z 393.744,A -85,B 0,C 180,E1 -12541.621,E2 -12541.621} C_VEL
LIN {X 0,Y 375.116,Z 393.762,A -85,B 0,C 180,E1 -12542.905,E2 -12542.905} C_VEL
LIN {X 0,Y 374.981,Z 396.958,A -85,B 0,C 180,E1 -12546.303,E2 -12546.303} C_VEL
LIN {X 0,Y 374.929,Z 400.34,A -85,B 0,C 180,E1 -12549.779,E2 -12549.779} C_VEL
LIN {X 0,Y 374.918,Z 400.472,A -85,B 0,C 180,E1 -12549.912,E2 -12549.912} C_VEL
LIN {X 0,Y 374.216,Z 401.128,A -85,B 0,C 180,E1 -12550.501,E2 -12550.501} C_VEL
LIN {X 0,Y 371.369,Z 402.318,A -85,B 0,C 180,E1 -12551.42,E2 -12551.42} C_VEL
LIN {X 0,Y 368.513,Z 403.518,A -85,B 0,C 180,E1 -12552.353,E2 -12552.353} C_VEL
LIN {X 0,Y 367.822,Z 404.18,A -85,B 0,C 180,E1 -12552.957,E2 -12552.957} C_VEL
LIN {X 0,Y 367.832,Z 404.371,A -85,B 0,C 180,E1 -12553.029,E2 -12553.029} C_VEL
LIN {X 0,Y 371.035,Z 417.818,A -85,B 0,C 180,E1 -12553.731,E2 -12553.731} C_VEL
LIN {X 0,Y 373.649,Z 430.389,A -85,B 0,C 180,E1 -12554.583,E2 -12554.583} C_VEL
LIN {X 0,Y 372.985,Z 441.622,A -85,B 0,C 180,E1 -12555.423,E2 -12555.423} C_VEL
LIN {X 0,Y 371.986,Z 453.848,A -85,B 0,C 180,E1 -12556.59,E2 -12556.59} C_VEL
LIN {X 0,Y 371.143,Z 464.162,A -85,B 0,C 180,E1 -12557.823,E2 -12557.823} C_VEL
LIN {X 0,Y 370.334,Z 473.763,A -85,B 0,C 180,E1 -12559.25,E2 -12559.25} C_VEL
LIN {X 0,Y 369.525,Z 482.152,A -85,B 0,C 180,E1 -12560.775,E2 -12560.775} C_VEL
LIN {X 0,Y 368.882,Z 489.545,A -85,B 0,C 180,E1 -12562.436,E2 -12562.436} C_VEL
LIN {X 0,Y 368.384,Z 495.386,A -85,B 0,C 180,E1 -12564.082,E2 -12564.082} C_VEL
LIN {X 0,Y 368.023,Z 500.077,A -85,B 0,C 180,E1 -12565.767,E2 -12565.767} C_VEL
LIN {X 0,Y 367.742,Z 503.963,A -85,B 0,C 180,E1 -12567.65,E2 -12567.65} C_VEL
LIN {X 0,Y 367.501,Z 506.386,A -85,B 0,C 180,E1 -12569.369,E2 -12569.369} C_VEL
LIN {X 0,Y 367.449,Z 508.028,A -85,B 0,C 180,E1 -12571.608,E2 -12571.608} C_VEL
LIN {X 0,Y 367.421,Z 508.19,A -85,B 0,C 180,E1 -12572.674,E2 -12572.674} C_VEL
LIN {X 0,Y 367.502,Z 507.883,A -85,B 0,C 180,E1 -12573.99,E2 -12573.99} C_VEL
LIN {X 0,Y 367.607,Z 507.165,A -85,B 0,C 180,E1 -12575.129,E2 -12575.129} C_VEL
LIN {X 0,Y 367.851,Z 505.689,A -85,B 0,C 180,E1 -12576.487,E2 -12576.487} C_VEL
LIN {X 0,Y 368.207,Z 503.027,A -85,B 0,C 180,E1 -12578.15,E2 -12578.15} C_VEL
LIN {X 0,Y 368.623,Z 499.046,A -85,B 0,C 180,E1 -12579.93,E2 -12579.93} C_VEL
LIN {X 0,Y 369.233,Z 494.001,A -85,B 0,C 180,E1 -12581.634,E2 -12581.634} C_VEL
LIN {X 0,Y 370.118,Z 487.045,A -85,B 0,C 180,E1 -12583.453,E2 -12583.453} C_VEL
LIN {X 0,Y 371.137,Z 478.797,A -85,B 0,C 180,E1 -12585.156,E2 -12585.156} C_VEL
LIN {X 0,Y 372.229,Z 469.934,A -85,B 0,C 180,E1 -12586.628,E2 -12586.628} C_VEL
LIN {X 0,Y 373.297,Z 460.443,A -85,B 0,C 180,E1 -12587.911,E2 -12587.911} C_VEL
LIN {X 0,Y 374.519,Z 448.722,A -85,B 0,C 180,E1 -12589.185,E2 -12589.185} C_VEL
LIN {X 0,Y 375.528,Z 437.186,A -85,B 0,C 180,E1 -12590.168,E2 -12590.168} C_VEL
LIN {X 0,Y 375.838,Z 433.631,A -85,B 0,C 180,E1 -12590.425,E2 -12590.425} C_VEL
LIN {X 0,Y 373.647,Z 423.724,A -85,B 0,C 180,E1 -12591.239,E2 -12591.239} C_VEL
LIN {X 0,Y 369.713,Z 411.362,A -85,B 0,C 180,E1 -12592.148,E2 -12592.148} C_VEL
LIN {X 0,Y 368.403,Z 407.238,A -85,B 0,C 180,E1 -12592.431,E2 -12592.431} C_VEL
LIN {X 0,Y 368.599,Z 405.52,A -85,B 0,C 180,E1 -12594.53,E2 -12594.53} C_VEL
LIN {X 0,Y 368.976,Z 401.315,A -85,B 0,C 180,E1 -12600.001,E2 -12600.001} C_VEL
LIN {X 0,Y 369.054,Z 399.73,A -85,B 0,C 180,E1 -12602.184,E2 -12602.184} C_VEL
LIN {X 0,Y 369.335,Z 396.792,A -85,B 0,C 180,E1 -12606.557,E2 -12606.557} C_VEL
LIN {X 0,Y 369.21,Z 395.453,A -85,B 0,C 180,E1 -12608.76,E2 -12608.76} C_VEL
LIN {X 0,Y 369.004,Z 394.522,A -85,B 0,C 180,E1 -12610.98,E2 -12610.98} C_VEL
LIN {X 0,Y 368.984,Z 394.524,A -85,B 0,C 180,E1 -12614.337,E2 -12614.337} C_VEL
LIN {X 0,Y 368.978,Z 394.525,A -85,B 0,C 180,E1 -12617.776,E2 -12617.776} C_VEL
LIN {X 0,Y 368.955,Z 394.525,A -85,B 0,C 180,E1 -12621.219,E2 -12621.219} C_VEL
LIN {X 0,Y 368.932,Z 394.529,A -85,B 0,C 180,E1 -12624.778,E2 -12624.778} C_VEL
LIN {X 0,Y 368.957,Z 394.528,A -85,B 0,C 180,E1 -12628.439,E2 -12628.439} C_VEL
LIN {X 0,Y 368.871,Z 394.537,A -85,B 0,C 180,E1 -12632.242,E2 -12632.242} C_VEL
LIN {X 0,Y 368.903,Z 394.535,A -85,B 0,C 180,E1 -12635.005,E2 -12635.005} C_VEL
LIN {X 0,Y 368.889,Z 394.535,A -85,B 0,C 180,E1 -12638.645,E2 -12638.645} C_VEL
LIN {X 0,Y 369.013,Z 395.014,A -85,B 0,C 180,E1 -12640.384,E2 -12640.384} C_VEL
LIN {X 0,Y 369.588,Z 397.969,A -85,B 0,C 180,E1 -12643.738,E2 -12643.738} C_VEL
LIN {X 0,Y 370.125,Z 401.352,A -85,B 0,C 180,E1 -12646.884,E2 -12646.884} C_VEL
LIN {X 0,Y 370.776,Z 405.089,A -85,B 0,C 180,E1 -12649.881,E2 -12649.881} C_VEL
LIN {X 0,Y 371.386,Z 409.108,A -85,B 0,C 180,E1 -12652.737,E2 -12652.737} C_VEL
LIN {X 0,Y 371.334,Z 411.844,A -85,B 0,C 180,E1 -12654.473,E2 -12654.473} C_VEL
LIN {X 0,Y 370.458,Z 417.805,A -85,B 0,C 180,E1 -12657.92,E2 -12657.92} C_VEL
LIN {X 0,Y 369.441,Z 425.85,A -85,B 0,C 180,E1 -12662.226,E2 -12662.226} C_VEL
LIN {X 0,Y 368.895,Z 431.798,A -85,B 0,C 180,E1 -12665.225,E2 -12665.225} C_VEL
LIN {X 0,Y 368.41,Z 439.107,A -85,B 0,C 180,E1 -12668.754,E2 -12668.754} C_VEL
LIN {X 0,Y 368.294,Z 440.763,A -85,B 0,C 180,E1 -12669.542,E2 -12669.542} C_VEL
LIN {X 0,Y 371.212,Z 454.581,A -85,B 0,C 180,E1 -12670.294,E2 -12670.294} C_VEL
LIN {X 0,Y 372.87,Z 466.301,A -85,B 0,C 180,E1 -12671.067,E2 -12671.067} C_VEL
LIN {X 0,Y 373.662,Z 479.05,A -85,B 0,C 180,E1 -12672.067,E2 -12672.067} C_VEL
LIN {X 0,Y 373.182,Z 486.889,A -85,B 0,C 180,E1 -12672.75,E2 -12672.75} C_VEL
LIN {X 0,Y 371.851,Z 498.526,A -85,B 0,C 180,E1 -12673.958,E2 -12673.958} C_VEL
LIN {X 0,Y 370.561,Z 509.553,A -85,B 0,C 180,E1 -12675.387,E2 -12675.387} C_VEL
LIN {X 0,Y 369.803,Z 518.399,A -85,B 0,C 180,E1 -12676.822,E2 -12676.822} C_VEL
LIN {X 0,Y 368.777,Z 526.724,A -85,B 0,C 180,E1 -12678.461,E2 -12678.461} C_VEL
LIN {X 0,Y 368.172,Z 533.486,A -85,B 0,C 180,E1 -12680.112,E2 -12680.112} C_VEL
LIN {X 0,Y 367.783,Z 538.915,A -85,B 0,C 180,E1 -12681.764,E2 -12681.764} C_VEL
LIN {X 0,Y 367.563,Z 543.171,A -85,B 0,C 180,E1 -12683.417,E2 -12683.417} C_VEL
LIN {X 0,Y 367.48,Z 545.409,A -85,B 0,C 180,E1 -12684.517,E2 -12684.517} C_VEL
LIN {X 0,Y 367.504,Z 547.197,A -85,B 0,C 180,E1 -12685.617,E2 -12685.617} C_VEL
LIN {X 0,Y 367.549,Z 549.532,A -85,B 0,C 180,E1 -12687.812,E2 -12687.812} C_VEL
LIN {X 0,Y 367.596,Z 550.04,A -85,B 0,C 180,E1 -12688.909,E2 -12688.909} C_VEL
LIN {X 0,Y 367.587,Z 550.138,A -85,B 0,C 180,E1 -12690.004,E2 -12690.004} C_VEL
LIN {X 0,Y 367.599,Z 549.839,A -85,B 0,C 180,E1 -12691.099,E2 -12691.099} C_VEL
LIN {X 0,Y 367.606,Z 549.129,A -85,B 0,C 180,E1 -12692.195,E2 -12692.195} C_VEL
LIN {X 0,Y 367.482,Z 547.947,A -85,B 0,C 180,E1 -12693.293,E2 -12693.293} C_VEL
LIN {X 0,Y 367.523,Z 545.399,A -85,B 0,C 180,E1 -12694.94,E2 -12694.94} C_VEL
LIN {X 0,Y 367.586,Z 541.795,A -85,B 0,C 180,E1 -12696.591,E2 -12696.591} C_VEL
LIN {X 0,Y 367.789,Z 537.05,A -85,B 0,C 180,E1 -12698.244,E2 -12698.244} C_VEL
LIN {X 0,Y 368.216,Z 529.895,A -85,B 0,C 180,E1 -12700.173,E2 -12700.173} C_VEL
LIN {X 0,Y 368.868,Z 522.108,A -85,B 0,C 180,E1 -12701.823,E2 -12701.823} C_VEL
LIN {X 0,Y 369.707,Z 512.361,A -85,B 0,C 180,E1 -12703.47,E2 -12703.47} C_VEL
LIN {X 0,Y 370.497,Z 502.753,A -85,B 0,C 180,E1 -12704.785,E2 -12704.785} C_VEL
LIN {X 0,Y 371.337,Z 492.408,A -85,B 0,C 180,E1 -12705.932,E2 -12705.932} C_VEL
LIN {X 0,Y 372.446,Z 480.08,A -85,B 0,C 180,E1 -12707.01,E2 -12707.01} C_VEL
LIN {X 0,Y 371.509,Z 468.799,A -85,B 0,C 180,E1 -12707.841,E2 -12707.841} C_VEL
LIN {X 0,Y 369.874,Z 455.593,A -85,B 0,C 180,E1 -12708.601,E2 -12708.601} C_VEL
LIN {X 0,Y 368.12,Z 443.536,A -85,B 0,C 180,E1 -12709.123,E2 -12709.123} C_VEL
LIN {X 0,Y 368.612,Z 435.254,A -85,B 0,C 180,E1 -12713.011,E2 -12713.011} C_VEL
LIN {X 0,Y 369.171,Z 427.925,A -85,B 0,C 180,E1 -12716.522,E2 -12716.522} C_VEL
LIN {X 0,Y 369.892,Z 420.338,A -85,B 0,C 180,E1 -12720.236,E2 -12720.236} C_VEL
LIN {X 0,Y 370.637,Z 413.938,A -85,B 0,C 180,E1 -12723.453,E2 -12723.453} C_VEL
LIN {X 0,Y 371.14,Z 409.115,A -85,B 0,C 180,E1 -12725.95,E2 -12725.95} C_VEL
LIN {X 0,Y 370.796,Z 405.307,A -85,B 0,C 180,E1 -12728.028,E2 -12728.028} C_VEL
LIN {X 0,Y 369.751,Z 398.948,A -85,B 0,C 180,E1 -12731.706,E2 -12731.706} C_VEL
LIN {X 0,Y 368.92,Z 394.53,A -85,B 0,C 180,E1 -12734.435,E2 -12734.435} C_VEL
LIN {X 0,Y 368.884,Z 394.537,A -85,B 0,C 180,E1 -12738.177,E2 -12738.177} C_VEL
LIN {X 0,Y 368.891,Z 394.536,A -85,B 0,C 180,E1 -12741.367,E2 -12741.367} C_VEL
LIN {X 0,Y 368.946,Z 394.53,A -85,B 0,C 180,E1 -12745.147,E2 -12745.147} C_VEL
LIN {X 0,Y 368.928,Z 394.532,A -85,B 0,C 180,E1 -12749.045,E2 -12749.045} C_VEL
LIN {X 0,Y 368.931,Z 394.53,A -85,B 0,C 180,E1 -12751.559,E2 -12751.559} C_VEL
LIN {X 0,Y 368.94,Z 394.53,A -85,B 0,C 180,E1 -12755.222,E2 -12755.222} C_VEL
LIN {X 0,Y 368.935,Z 394.532,A -85,B 0,C 180,E1 -12758.981,E2 -12758.981} C_VEL
LIN {X 0,Y 369.007,Z 394.518,A -85,B 0,C 180,E1 -12762.257,E2 -12762.257} C_VEL
LIN {X 0,Y 369.052,Z 394.512,A -85,B 0,C 180,E1 -12766.228,E2 -12766.228} C_VEL
LIN {X 0,Y 369.076,Z 394.509,A -85,B 0,C 180,E1 -12770.131,E2 -12770.131} C_VEL
LIN {X 0,Y 369.193,Z 394.496,A -85,B 0,C 180,E1 -12773.441,E2 -12773.441} C_VEL
LIN {X 0,Y 369.327,Z 394.478,A -85,B 0,C 180,E1 -12777.818,E2 -12777.818} C_VEL
LIN {X 0,Y 369.444,Z 394.463,A -85,B 0,C 180,E1 -12779.999,E2 -12779.999} C_VEL
LIN {X 0,Y 369.32,Z 394.479,A -85,B 0,C 180,E1 -12782.18,E2 -12782.18} C_VEL
LIN {X 0,Y 369.172,Z 394.5,A -85,B 0,C 180,E1 -12786.558,E2 -12786.558} C_VEL
LIN {X 0,Y 369.074,Z 394.509,A -85,B 0,C 180,E1 -12789.867,E2 -12789.867} C_VEL
LIN {X 0,Y 369.049,Z 394.513,A -85,B 0,C 180,E1 -12793.77,E2 -12793.77} C_VEL
LIN {X 0,Y 369.003,Z 394.518,A -85,B 0,C 180,E1 -12797.741,E2 -12797.741} C_VEL
LIN {X 0,Y 368.921,Z 394.53,A -85,B 0,C 180,E1 -12801.219,E2 -12801.219} C_VEL
LIN {X 0,Y 368.963,Z 394.527,A -85,B 0,C 180,E1 -12804.774,E2 -12804.774} C_VEL
LIN {X 0,Y 368.972,Z 394.523,A -85,B 0,C 180,E1 -12807.201,E2 -12807.201} C_VEL
LIN {X 0,Y 368.92,Z 394.531,A -85,B 0,C 180,E1 -12810.985,E2 -12810.985} C_VEL
LIN {X 0,Y 368.944,Z 394.529,A -85,B 0,C 180,E1 -12814.851,E2 -12814.851} C_VEL
LIN {X 0,Y 368.889,Z 394.537,A -85,B 0,C 180,E1 -12818.632,E2 -12818.632} C_VEL
LIN {X 0,Y 368.886,Z 394.534,A -85,B 0,C 180,E1 -12822.006,E2 -12822.006} C_VEL
LIN {X 0,Y 368.885,Z 394.534,A -85,B 0,C 180,E1 -12825.173,E2 -12825.173} C_VEL
LIN {X 0,Y 368.885,Z 394.536,A -85,B 0,C 180,E1 -12828.174,E2 -12828.174} C_VEL
LIN {X 0,Y 368.907,Z 394.53,A -85,B 0,C 180,E1 -12831.358,E2 -12831.358} C_VEL
LIN {X 0,Y 368.941,Z 394.527,A -85,B 0,C 180,E1 -12835.143,E2 -12835.143} C_VEL
LIN {X 0,Y 368.933,Z 394.528,A -85,B 0,C 180,E1 -12839.043,E2 -12839.043} C_VEL
LIN {X 0,Y 368.965,Z 394.525,A -85,B 0,C 180,E1 -12842.793,E2 -12842.793} C_VEL
LIN {X 0,Y 368.947,Z 394.529,A -85,B 0,C 180,E1 -12846.109,E2 -12846.109} C_VEL
LIN {X 0,Y 368.937,Z 394.529,A -85,B 0,C 180,E1 -12849.943,E2 -12849.943} C_VEL
LIN {X 0,Y 368.974,Z 394.521,A -85,B 0,C 180,E1 -12853.395,E2 -12853.395} C_VEL
LIN {X 0,Y 369.056,Z 394.513,A -85,B 0,C 180,E1 -12856.786,E2 -12856.786} C_VEL
LIN {X 0,Y 369.064,Z 394.515,A -85,B 0,C 180,E1 -12860.128,E2 -12860.128} C_VEL
LIN {X 0,Y 369.194,Z 394.495,A -85,B 0,C 180,E1 -12863.438,E2 -12863.438} C_VEL
LIN {X 0,Y 369.31,Z 394.483,A -85,B 0,C 180,E1 -12867.815,E2 -12867.815} C_VEL
LIN {X 0,Y 369.449,Z 394.467,A -85,B 0,C 180,E1 -12869.996,E2 -12869.996} C_VEL
LIN {X 0,Y 369.311,Z 394.484,A -85,B 0,C 180,E1 -12872.177,E2 -12872.177} C_VEL
LIN {X 0,Y 369.198,Z 394.496,A -85,B 0,C 180,E1 -12876.554,E2 -12876.554} C_VEL
LIN {X 0,Y 369.128,Z 394.504,A -85,B 0,C 180,E1 -12878.757,E2 -12878.757} C_VEL
LIN {X 0,Y 369.001,Z 394.524,A -85,B 0,C 180,E1 -12882.089,E2 -12882.089} C_VEL
LIN {X 0,Y 368.987,Z 394.521,A -85,B 0,C 180,E1 -12885.461,E2 -12885.461} C_VEL
LIN {X 0,Y 368.966,Z 394.523,A -85,B 0,C 180,E1 -12888.889,E2 -12888.889} C_VEL
LIN {X 0,Y 368.913,Z 394.532,A -85,B 0,C 180,E1 -12892.391,E2 -12892.391} C_VEL
LIN {X 0,Y 368.897,Z 394.536,A -85,B 0,C 180,E1 -12895.983,E2 -12895.983} C_VEL
LIN {X 0,Y 368.51,Z 394.585,A -85,B 0,C 180,E1 -12899.721,E2 -12899.721} C_VEL
LIN {X 0,Y 368.082,Z 394.638,A -85,B 0,C 180,E1 -12902.85,E2 -12902.85} C_VEL
LIN {X 0,Y 367.926,Z 397.693,A -85,B 0,C 180,E1 -12906.303,E2 -12906.303} C_VEL
LIN {X 0,Y 367.841,Z 401.153,A -85,B 0,C 180,E1 -12909.892,E2 -12909.892} C_VEL
LIN {X 0,Y 367.822,Z 404.18,A -85,B 0,C 180,E1 -12912.957,E2 -12912.957} C_VEL
LIN {X 0,Y 368.517,Z 404.504,A -85,B 0,C 180,E1 -12913.065,E2 -12913.065} C_VEL
LIN {X 0,Y 373.346,Z 406.844,A -85,B 0,C 180,E1 -12913.356,E2 -12913.356} C_VEL
LIN {X 0,Y 375.103,Z 408.879,A -85,B 0,C 180,E1 -12913.516,E2 -12913.516} C_VEL
LIN {X 0,Y 375.278,Z 410.93,A -85,B 0,C 180,E1 -12913.593,E2 -12913.593} C_VEL
LIN {X 0,Y 374.117,Z 412.854,A -85,B 0,C 180,E1 -12913.61,E2 -12913.61} C_VEL
LIN {X 0,Y 368.66,Z 417.515,A -85,B 0,C 180,E1 -12913.609,E2 -12913.609} C_VEL
LIN {X 0,Y 367.818,Z 419.724,A -85,B 0,C 180,E1 -12913.68,E2 -12913.68} C_VEL
LIN {X 0,Y 367.457,Z 427.174,A -85,B 0,C 180,E1 -12914.104,E2 -12914.104} C_VEL
LIN {X 0,Y 366.626,Z 434.081,A -85,B 0,C 180,E1 -12914.548,E2 -12914.548} C_VEL
LIN {X 0,Y 365.822,Z 446.062,A -85,B 0,C 180,E1 -12915.531,E2 -12915.531} C_VEL
LIN {X 0,Y 364.799,Z 457.474,A -85,B 0,C 180,E1 -12916.726,E2 -12916.726} C_VEL
LIN {X 0,Y 363.93,Z 467.547,A -85,B 0,C 180,E1 -12918.038,E2 -12918.038} C_VEL
LIN {X 0,Y 363.075,Z 477.117,A -85,B 0,C 180,E1 -12919.576,E2 -12919.576} C_VEL
LIN {X 0,Y 362.253,Z 485.397,A -85,B 0,C 180,E1 -12921.233,E2 -12921.233} C_VEL
LIN {X 0,Y 361.627,Z 492.316,A -85,B 0,C 180,E1 -12922.955,E2 -12922.955} C_VEL
LIN {X 0,Y 361.139,Z 498.177,A -85,B 0,C 180,E1 -12924.81,E2 -12924.81} C_VEL
LIN {X 0,Y 360.807,Z 502.995,A -85,B 0,C 180,E1 -12926.875,E2 -12926.875} C_VEL
LIN {X 0,Y 360.447,Z 506.465,A -85,B 0,C 180,E1 -12929.072,E2 -12929.072} C_VEL
LIN {X 0,Y 360.361,Z 508.298,A -85,B 0,C 180,E1 -12931.345,E2 -12931.345} C_VEL
LIN {X 0,Y 360.362,Z 508.566,A -85,B 0,C 180,E1 -12933.35,E2 -12933.35} C_VEL
LIN {X 0,Y 360.463,Z 508.043,A -85,B 0,C 180,E1 -12934.601,E2 -12934.601} C_VEL
LIN {X 0,Y 360.743,Z 506.565,A -85,B 0,C 180,E1 -12936.285,E2 -12936.285} C_VEL
LIN {X 0,Y 361.191,Z 503.524,A -85,B 0,C 180,E1 -12938.304,E2 -12938.304} C_VEL
LIN {X 0,Y 361.637,Z 499.565,A -85,B 0,C 180,E1 -12940.119,E2 -12940.119} C_VEL
LIN {X 0,Y 362.313,Z 494.336,A -85,B 0,C 180,E1 -12941.92,E2 -12941.92} C_VEL
LIN {X 0,Y 363.236,Z 487.627,A -85,B 0,C 180,E1 -12943.708,E2 -12943.708} C_VEL
LIN {X 0,Y 364.321,Z 479.273,A -85,B 0,C 180,E1 -12945.478,E2 -12945.478} C_VEL
LIN {X 0,Y 365.465,Z 470.673,A -85,B 0,C 180,E1 -12946.942,E2 -12946.942} C_VEL
LIN {X 0,Y 366.696,Z 460.424,A -85,B 0,C 180,E1 -12948.347,E2 -12948.347} C_VEL
LIN {X 0,Y 367.874,Z 449.588,A -85,B 0,C 180,E1 -12949.544,E2 -12949.544} C_VEL
LIN {X 0,Y 368.928,Z 438.612,A -85,B 0,C 180,E1 -12950.511,E2 -12950.511} C_VEL
LIN {X 0,Y 369.229,Z 435.074,A -85,B 0,C 180,E1 -12950.774,E2 -12950.774} C_VEL
LIN {X 0,Y 366.802,Z 424.306,A -85,B 0,C 180,E1 -12951.704,E2 -12951.704} C_VEL
LIN {X 0,Y 363.026,Z 412.661,A -85,B 0,C 180,E1 -12952.616,E2 -12952.616} C_VEL
LIN {X 0,Y 361.414,Z 407.761,A -85,B 0,C 180,E1 -12952.951,E2 -12952.951} C_VEL
LIN {X 0,Y 361.534,Z 405.737,A -85,B 0,C 180,E1 -12955.541,E2 -12955.541} C_VEL
LIN {X 0,Y 361.951,Z 402.387,A -85,B 0,C 180,E1 -12960.001,E2 -12960.001} C_VEL
LIN {X 0,Y 362.043,Z 400.822,A -85,B 0,C 180,E1 -12962.226,E2 -12962.226} C_VEL
LIN {X 0,Y 362.328,Z 397.893,A -85,B 0,C 180,E1 -12966.684,E2 -12966.684} C_VEL
LIN {X 0,Y 362.197,Z 396.598,A -85,B 0,C 180,E1 -12968.931,E2 -12968.931} C_VEL
LIN {X 0,Y 361.952,Z 395.41,A -85,B 0,C 180,E1 -12971.197,E2 -12971.197} C_VEL
LIN {X 0,Y 361.933,Z 395.403,A -85,B 0,C 180,E1 -12974.623,E2 -12974.623} C_VEL
LIN {X 0,Y 361.933,Z 395.401,A -85,B 0,C 180,E1 -12978.102,E2 -12978.102} C_VEL
LIN {X 0,Y 361.9,Z 395.405,A -85,B 0,C 180,E1 -12981.653,E2 -12981.653} C_VEL
LIN {X 0,Y 361.9,Z 395.408,A -85,B 0,C 180,E1 -12985.293,E2 -12985.293} C_VEL
LIN {X 0,Y 361.893,Z 395.405,A -85,B 0,C 180,E1 -12987.781,E2 -12987.781} C_VEL
LIN {X 0,Y 361.819,Z 395.415,A -85,B 0,C 180,E1 -12991.289,E2 -12991.289} C_VEL
LIN {X 0,Y 361.828,Z 395.414,A -85,B 0,C 180,E1 -12994.284,E2 -12994.284} C_VEL
LIN {X 0,Y 361.841,Z 395.413,A -85,B 0,C 180,E1 -12997.227,E2 -12997.227} C_VEL
LIN {X 0,Y 361.879,Z 395.666,A -85,B 0,C 180,E1 -12999.037,E2 -12999.037} C_VEL
LIN {X 0,Y 362.453,Z 398.447,A -85,B 0,C 180,E1 -13002.547,E2 -13002.547} C_VEL
LIN {X 0,Y 363.009,Z 401.692,A -85,B 0,C 180,E1 -13005.823,E2 -13005.823} C_VEL
LIN {X 0,Y 363.638,Z 405.295,A -85,B 0,C 180,E1 -13008.927,E2 -13008.927} C_VEL
LIN {X 0,Y 364.342,Z 409.77,A -85,B 0,C 180,E1 -13012.268,E2 -13012.268} C_VEL
LIN {X 0,Y 364.434,Z 412.514,A -85,B 0,C 180,E1 -13014.093,E2 -13014.093} C_VEL
LIN {X 0,Y 363.604,Z 417.768,A -85,B 0,C 180,E1 -13017.24,E2 -13017.24} C_VEL
LIN {X 0,Y 362.618,Z 424.579,A -85,B 0,C 180,E1 -13021.024,E2 -13021.024} C_VEL
LIN {X 0,Y 362.056,Z 430.441,A -85,B 0,C 180,E1 -13024.108,E2 -13024.108} C_VEL
LIN {X 0,Y 361.487,Z 437.648,A -85,B 0,C 180,E1 -13027.726,E2 -13027.726} C_VEL
LIN {X 0,Y 361.327,Z 440.389,A -85,B 0,C 180,E1 -13029.009,E2 -13029.009} C_VEL
LIN {X 0,Y 364.37,Z 454.382,A -85,B 0,C 180,E1 -13029.822,E2 -13029.822} C_VEL
LIN {X 0,Y 366.083,Z 466.197,A -85,B 0,C 180,E1 -13030.636,E2 -13030.636} C_VEL
LIN {X 0,Y 366.851,Z 477.939,A -85,B 0,C 180,E1 -13031.578,E2 -13031.578} C_VEL
LIN {X 0,Y 366.607,Z 485.843,A -85,B 0,C 180,E1 -13032.287,E2 -13032.287} C_VEL
LIN {X 0,Y 365.19,Z 497.556,A -85,B 0,C 180,E1 -13033.514,E2 -13033.514} C_VEL
LIN {X 0,Y 363.898,Z 507.784,A -85,B 0,C 180,E1 -13034.845,E2 -13034.845} C_VEL
LIN {X 0,Y 363.012,Z 516.775,A -85,B 0,C 180,E1 -13036.285,E2 -13036.285} C_VEL
LIN {X 0,Y 361.984,Z 525.314,A -85,B 0,C 180,E1 -13037.958,E2 -13037.958} C_VEL
LIN {X 0,Y 361.262,Z 532.249,A -85,B 0,C 180,E1 -13039.638,E2 -13039.638} C_VEL
LIN {X 0,Y 360.735,Z 538.676,A -85,B 0,C 180,E1 -13041.602,E2 -13041.602} C_VEL
LIN {X 0,Y 360.497,Z 542.89,A -85,B 0,C 180,E1 -13043.287,E2 -13043.287} C_VEL
LIN {X 0,Y 360.394,Z 545.087,A -85,B 0,C 180,E1 -13044.409,E2 -13044.409} C_VEL
LIN {X 0,Y 360.408,Z 546.854,A -85,B 0,C 180,E1 -13045.531,E2 -13045.531} C_VEL
LIN {X 0,Y 360.366,Z 548.206,A -85,B 0,C 180,E1 -13046.65,E2 -13046.65} C_VEL
LIN {X 0,Y 360.449,Z 549.143,A -85,B 0,C 180,E1 -13047.769,E2 -13047.769} C_VEL
LIN {X 0,Y 360.529,Z 549.633,A -85,B 0,C 180,E1 -13048.887,E2 -13048.887} C_VEL
LIN {X 0,Y 360.521,Z 549.717,A -85,B 0,C 180,E1 -13050.004,E2 -13050.004} C_VEL
LIN {X 0,Y 360.534,Z 549.402,A -85,B 0,C 180,E1 -13051.121,E2 -13051.121} C_VEL
LIN {X 0,Y 360.507,Z 548.659,A -85,B 0,C 180,E1 -13052.239,E2 -13052.239} C_VEL
LIN {X 0,Y 360.396,Z 547.456,A -85,B 0,C 180,E1 -13053.358,E2 -13053.358} C_VEL
LIN {X 0,Y 360.445,Z 544.868,A -85,B 0,C 180,E1 -13055.038,E2 -13055.038} C_VEL
LIN {X 0,Y 360.512,Z 541.222,A -85,B 0,C 180,E1 -13056.721,E2 -13056.721} C_VEL
LIN {X 0,Y 360.739,Z 536.431,A -85,B 0,C 180,E1 -13058.406,E2 -13058.406} C_VEL
LIN {X 0,Y 361.117,Z 530.353,A -85,B 0,C 180,E1 -13060.092,E2 -13060.092} C_VEL
LIN {X 0,Y 361.739,Z 522.787,A -85,B 0,C 180,E1 -13061.775,E2 -13061.775} C_VEL
LIN {X 0,Y 362.397,Z 515.067,A -85,B 0,C 180,E1 -13063.175,E2 -13063.175} C_VEL
LIN {X 0,Y 363.223,Z 505.046,A -85,B 0,C 180,E1 -13064.656,E2 -13064.656} C_VEL
LIN {X 0,Y 364.272,Z 494.046,A -85,B 0,C 180,E1 -13065.961,E2 -13065.961} C_VEL
LIN {X 0,Y 365.338,Z 482.303,A -85,B 0,C 180,E1 -13067.063,E2 -13067.063} C_VEL
LIN {X 0,Y 365.262,Z 476.935,A -85,B 0,C 180,E1 -13067.5,E2 -13067.5} C_VEL
LIN {X 0,Y 363.997,Z 464.226,A -85,B 0,C 180,E1 -13068.396,E2 -13068.396} C_VEL
LIN {X 0,Y 362.222,Z 451.158,A -85,B 0,C 180,E1 -13069.107,E2 -13069.107} C_VEL
LIN {X 0,Y 361.085,Z 443.191,A -85,B 0,C 180,E1 -13069.437,E2 -13069.437} C_VEL
LIN {X 0,Y 361.619,Z 434.838,A -85,B 0,C 180,E1 -13073.461,E2 -13073.461} C_VEL
LIN {X 0,Y 362.145,Z 428.05,A -85,B 0,C 180,E1 -13076.784,E2 -13076.784} C_VEL
LIN {X 0,Y 362.83,Z 421.149,A -85,B 0,C 180,E1 -13080.243,E2 -13080.243} C_VEL
LIN {X 0,Y 363.645,Z 414.242,A -85,B 0,C 180,E1 -13083.793,E2 -13083.793} C_VEL
LIN {X 0,Y 364.113,Z 410.36,A -85,B 0,C 180,E1 -13085.837,E2 -13085.837} C_VEL
LIN {X 0,Y 363.898,Z 407.118,A -85,B 0,C 180,E1 -13087.641,E2 -13087.641} C_VEL
LIN {X 0,Y 362.966,Z 401.421,A -85,B 0,C 180,E1 -13090.961,E2 -13090.961} C_VEL
LIN {X 0,Y 361.88,Z 395.444,A -85,B 0,C 180,E1 -13094.655,E2 -13094.655} C_VEL
LIN {X 0,Y 361.845,Z 395.413,A -85,B 0,C 180,E1 -13097.571,E2 -13097.571} C_VEL
LIN {X 0,Y 361.858,Z 395.411,A -85,B 0,C 180,E1 -13101.573,E2 -13101.573} C_VEL
LIN {X 0,Y 361.885,Z 395.406,A -85,B 0,C 180,E1 -13104.657,E2 -13104.657} C_VEL
LIN {X 0,Y 361.853,Z 395.409,A -85,B 0,C 180,E1 -13108.371,E2 -13108.371} C_VEL
LIN {X 0,Y 361.882,Z 395.409,A -85,B 0,C 180,E1 -13110.953,E2 -13110.953} C_VEL
LIN {X 0,Y 361.898,Z 395.405,A -85,B 0,C 180,E1 -13114.707,E2 -13114.707} C_VEL
LIN {X 0,Y 361.876,Z 395.406,A -85,B 0,C 180,E1 -13118.345,E2 -13118.345} C_VEL
LIN {X 0,Y 361.936,Z 395.398,A -85,B 0,C 180,E1 -13122.085,E2 -13122.085} C_VEL
LIN {X 0,Y 361.976,Z 395.396,A -85,B 0,C 180,E1 -13125.379,E2 -13125.379} C_VEL
LIN {X 0,Y 361.983,Z 395.397,A -85,B 0,C 180,E1 -13128.804,E2 -13128.804} C_VEL
LIN {X 0,Y 362.108,Z 395.377,A -85,B 0,C 180,E1 -13132.191,E2 -13132.191} C_VEL
LIN {X 0,Y 362.117,Z 395.377,A -85,B 0,C 180,E1 -13134.43,E2 -13134.43} C_VEL
LIN {X 0,Y 362.291,Z 395.354,A -85,B 0,C 180,E1 -13137.776,E2 -13137.776} C_VEL
LIN {X 0,Y 362.394,Z 395.341,A -85,B 0,C 180,E1 -13139.999,E2 -13139.999} C_VEL
LIN {X 0,Y 362.283,Z 395.356,A -85,B 0,C 180,E1 -13142.223,E2 -13142.223} C_VEL
LIN {X 0,Y 362.135,Z 395.378,A -85,B 0,C 180,E1 -13146.686,E2 -13146.686} C_VEL
LIN {X 0,Y 362.011,Z 395.389,A -85,B 0,C 180,E1 -13150.062,E2 -13150.062} C_VEL
LIN {X 0,Y 362.01,Z 395.389,A -85,B 0,C 180,E1 -13153.897,E2 -13153.897} C_VEL
LIN {X 0,Y 361.939,Z 395.402,A -85,B 0,C 180,E1 -13156.933,E2 -13156.933} C_VEL
LIN {X 0,Y 361.894,Z 395.407,A -85,B 0,C 180,E1 -13160.459,E2 -13160.459} C_VEL
LIN {X 0,Y 361.904,Z 395.403,A -85,B 0,C 180,E1 -13164.111,E2 -13164.111} C_VEL
LIN {X 0,Y 361.951,Z 395.402,A -85,B 0,C 180,E1 -13166.719,E2 -13166.719} C_VEL
LIN {X 0,Y 361.869,Z 395.41,A -85,B 0,C 180,E1 -13170.327,E2 -13170.327} C_VEL
LIN {X 0,Y 361.863,Z 395.411,A -85,B 0,C 180,E1 -13174.278,E2 -13174.278} C_VEL
LIN {X 0,Y 361.869,Z 395.408,A -85,B 0,C 180,E1 -13177.22,E2 -13177.22} C_VEL
LIN {X 0,Y 361.84,Z 395.414,A -85,B 0,C 180,E1 -13180.752,E2 -13180.752} C_VEL
LIN {X 0,Y 361.823,Z 395.416,A -85,B 0,C 180,E1 -13184.366,E2 -13184.366} C_VEL
LIN {X 0,Y 361.84,Z 395.41,A -85,B 0,C 180,E1 -13187.566,E2 -13187.566} C_VEL
LIN {X 0,Y 361.868,Z 395.409,A -85,B 0,C 180,E1 -13190.972,E2 -13190.972} C_VEL
LIN {X 0,Y 361.878,Z 395.41,A -85,B 0,C 180,E1 -13194.652,E2 -13194.652} C_VEL
LIN {X 0,Y 361.841,Z 395.415,A -85,B 0,C 180,E1 -13198.367,E2 -13198.367} C_VEL
LIN {X 0,Y 361.911,Z 395.406,A -85,B 0,C 180,E1 -13202.218,E2 -13202.218} C_VEL
LIN {X 0,Y 361.93,Z 395.402,A -85,B 0,C 180,E1 -13204.706,E2 -13204.706} C_VEL
LIN {X 0,Y 361.893,Z 395.409,A -85,B 0,C 180,E1 -13208.343,E2 -13208.343} C_VEL
LIN {X 0,Y 361.967,Z 395.398,A -85,B 0,C 180,E1 -13212.058,E2 -13212.058} C_VEL
LIN {X 0,Y 361.996,Z 395.395,A -85,B 0,C 180,E1 -13216.097,E2 -13216.097} C_VEL
LIN {X 0,Y 362.028,Z 395.39,A -85,B 0,C 180,E1 -13219.934,E2 -13219.934} C_VEL
LIN {X 0,Y 362.156,Z 395.371,A -85,B 0,C 180,E1 -13223.31,E2 -13223.31} C_VEL
LIN {X 0,Y 362.274,Z 395.359,A -85,B 0,C 180,E1 -13227.772,E2 -13227.772} C_VEL
LIN {X 0,Y 362.419,Z 395.342,A -85,B 0,C 180,E1 -13229.996,E2 -13229.996} C_VEL
LIN {X 0,Y 362.275,Z 395.361,A -85,B 0,C 180,E1 -13232.219,E2 -13232.219} C_VEL
LIN {X 0,Y 362.162,Z 395.371,A -85,B 0,C 180,E1 -13236.682,E2 -13236.682} C_VEL
LIN {X 0,Y 362.064,Z 395.383,A -85,B 0,C 180,E1 -13238.929,E2 -13238.929} C_VEL
LIN {X 0,Y 361.954,Z 395.4,A -85,B 0,C 180,E1 -13242.328,E2 -13242.328} C_VEL
LIN {X 0,Y 361.949,Z 395.398,A -85,B 0,C 180,E1 -13244.616,E2 -13244.616} C_VEL
LIN {X 0,Y 361.943,Z 395.402,A -85,B 0,C 180,E1 -13248.095,E2 -13248.095} C_VEL
LIN {X 0,Y 361.874,Z 395.409,A -85,B 0,C 180,E1 -13251.649,E2 -13251.649} C_VEL
LIN {X 0,Y 361.86,Z 395.408,A -85,B 0,C 180,E1 -13255.29,E2 -13255.29} C_VEL
LIN {X 0,Y 361.662,Z 395.437,A -85,B 0,C 180,E1 -13257.794,E2 -13257.794} C_VEL
LIN {X 0,Y 361.238,Z 395.488,A -85,B 0,C 180,E1 -13261.128,E2 -13261.128} C_VEL
LIN {X 0,Y 360.984,Z 395.523,A -85,B 0,C 180,E1 -13263.16,E2 -13263.16} C_VEL
LIN {X 0,Y 360.859,Z 399.199,A -85,B 0,C 180,E1 -13267.132,E2 -13267.132} C_VEL
LIN {X 0,Y 360.76,Z 402.502,A -85,B 0,C 180,E1 -13270.559,E2 -13270.559} C_VEL
LIN {X 0,Y 360.774,Z 404.74,A -85,B 0,C 180,E1 -13272.722,E2 -13272.722} C_VEL
LIN {X 0,Y 363.974,Z 418.336,A -85,B 0,C 180,E1 -13273.443,E2 -13273.443} C_VEL
LIN {X 0,Y 366.544,Z 430.185,A -85,B 0,C 180,E1 -13274.263,E2 -13274.263} C_VEL
LIN {X 0,Y 366.708,Z 432.769,A -85,B 0,C 180,E1 -13274.454,E2 -13274.454} C_VEL
LIN {X 0,Y 366.626,Z 434.081,A -85,B 0,C 180,E1 -13274.548,E2 -13274.548} C_VEL
LIN {X 0,Y 365.64,Z 439.42,A -85,B 0,C 180,E1 -13274.925,E2 -13274.925} C_VEL
LIN {X 0,Y 362.202,Z 447.795,A -85,B 0,C 180,E1 -13275.556,E2 -13275.556} C_VEL
LIN {X 0,Y 358.701,Z 455.842,A -85,B 0,C 180,E1 -13276.291,E2 -13276.291} C_VEL
LIN {X 0,Y 357.607,Z 460.555,A -85,B 0,C 180,E1 -13276.835,E2 -13276.835} C_VEL
LIN {X 0,Y 356.683,Z 470.764,A -85,B 0,C 180,E1 -13278.273,E2 -13278.273} C_VEL
LIN {X 0,Y 355.758,Z 480.313,A -85,B 0,C 180,E1 -13279.941,E2 -13279.941} C_VEL
LIN {X 0,Y 355.081,Z 487.249,A -85,B 0,C 180,E1 -13281.432,E2 -13281.432} C_VEL
LIN {X 0,Y 354.542,Z 493.042,A -85,B 0,C 180,E1 -13282.945,E2 -13282.945} C_VEL
LIN {X 0,Y 354.043,Z 498.858,A -85,B 0,C 180,E1 -13284.855,E2 -13284.855} C_VEL
LIN {X 0,Y 353.779,Z 502.797,A -85,B 0,C 180,E1 -13286.538,E2 -13286.538} C_VEL
LIN {X 0,Y 353.389,Z 506.469,A -85,B 0,C 180,E1 -13288.766,E2 -13288.766} C_VEL
LIN {X 0,Y 353.284,Z 508.553,A -85,B 0,C 180,E1 -13291.069,E2 -13291.069} C_VEL
LIN {X 0,Y 353.291,Z 508.979,A -85,B 0,C 180,E1 -13293.519,E2 -13293.519} C_VEL
LIN {X 0,Y 353.48,Z 508.084,A -85,B 0,C 180,E1 -13295.323,E2 -13295.323} C_VEL
LIN {X 0,Y 353.732,Z 506.818,A -85,B 0,C 180,E1 -13296.588,E2 -13296.588} C_VEL
LIN {X 0,Y 354.011,Z 505.093,A -85,B 0,C 180,E1 -13297.841,E2 -13297.841} C_VEL
LIN {X 0,Y 354.478,Z 501.564,A -85,B 0,C 180,E1 -13299.7,E2 -13299.7} C_VEL
LIN {X 0,Y 355.2,Z 496.196,A -85,B 0,C 180,E1 -13301.737,E2 -13301.737} C_VEL
LIN {X 0,Y 356.195,Z 489.485,A -85,B 0,C 180,E1 -13303.672,E2 -13303.672} C_VEL
LIN {X 0,Y 357.3,Z 481.479,A -85,B 0,C 180,E1 -13305.477,E2 -13305.477} C_VEL
LIN {X 0,Y 358.48,Z 473.211,A -85,B 0,C 180,E1 -13306.971,E2 -13306.971} C_VEL
LIN {X 0,Y 359.637,Z 463.953,A -85,B 0,C 180,E1 -13308.347,E2 -13308.347} C_VEL
LIN {X 0,Y 360.976,Z 453.271,A -85,B 0,C 180,E1 -13309.626,E2 -13309.626} C_VEL
LIN {X 0,Y 362.25,Z 440.982,A -85,B 0,C 180,E1 -13310.791,E2 -13310.791} C_VEL
LIN {X 0,Y 362.604,Z 436.174,A -85,B 0,C 180,E1 -13311.177,E2 -13311.177} C_VEL
LIN {X 0,Y 360.387,Z 426.444,A -85,B 0,C 180,E1 -13312.066,E2 -13312.066} C_VEL
LIN {X 0,Y 356.531,Z 414.198,A -85,B 0,C 180,E1 -13313.074,E2 -13313.074} C_VEL
LIN {X 0,Y 354.485,Z 408.721,A -85,B 0,C 180,E1 -13313.491,E2 -13313.491} C_VEL
LIN {X 0,Y 354.441,Z 408.286,A -85,B 0,C 180,E1 -13313.526,E2 -13313.526} C_VEL
LIN {X 0,Y 354.435,Z 405.978,A -85,B 0,C 180,E1 -13316.591,E2 -13316.591} C_VEL
LIN {X 0,Y 354.925,Z 403.464,A -85,B 0,C 180,E1 -13320.001,E2 -13320.001} C_VEL
LIN {X 0,Y 355.031,Z 401.921,A -85,B 0,C 180,E1 -13322.27,E2 -13322.27} C_VEL
LIN {X 0,Y 355.329,Z 399.04,A -85,B 0,C 180,E1 -13326.816,E2 -13326.816} C_VEL
LIN {X 0,Y 355.183,Z 397.771,A -85,B 0,C 180,E1 -13329.109,E2 -13329.109} C_VEL
LIN {X 0,Y 354.896,Z 396.281,A -85,B 0,C 180,E1 -13332.583,E2 -13332.583} C_VEL
LIN {X 0,Y 354.873,Z 396.283,A -85,B 0,C 180,E1 -13336.098,E2 -13336.098} C_VEL
LIN {X 0,Y 354.881,Z 396.28,A -85,B 0,C 180,E1 -13338.474,E2 -13338.474} C_VEL
LIN {X 0,Y 354.86,Z 396.285,A -85,B 0,C 180,E1 -13342.105,E2 -13342.105} C_VEL
LIN {X 0,Y 354.871,Z 396.28,A -85,B 0,C 180,E1 -13345.831,E2 -13345.831} C_VEL
LIN {X 0,Y 354.826,Z 396.285,A -85,B 0,C 180,E1 -13349.682,E2 -13349.682} C_VEL
LIN {X 0,Y 354.78,Z 396.293,A -85,B 0,C 180,E1 -13353.706,E2 -13353.706} C_VEL
LIN {X 0,Y 354.775,Z 396.296,A -85,B 0,C 180,E1 -13356.463,E2 -13356.463} C_VEL
LIN {X 0,Y 354.819,Z 396.556,A -85,B 0,C 180,E1 -13357.882,E2 -13357.882} C_VEL
LIN {X 0,Y 355.35,Z 398.971,A -85,B 0,C 180,E1 -13361.284,E2 -13361.284} C_VEL
LIN {X 0,Y 355.864,Z 402.067,A -85,B 0,C 180,E1 -13364.694,E2 -13364.694} C_VEL
LIN {X 0,Y 356.586,Z 406.256,A -85,B 0,C 180,E1 -13368.5,E2 -13368.5} C_VEL
LIN {X 0,Y 357.304,Z 410.592,A -85,B 0,C 180,E1 -13371.887,E2 -13371.887} C_VEL
LIN {X 0,Y 357.455,Z 413.464,A -85,B 0,C 180,E1 -13373.861,E2 -13373.861} C_VEL
LIN {X 0,Y 356.77,Z 417.771,A -85,B 0,C 180,E1 -13376.531,E2 -13376.531} C_VEL
